ABB RobotStudio station: OP70 Robot Program.rspag

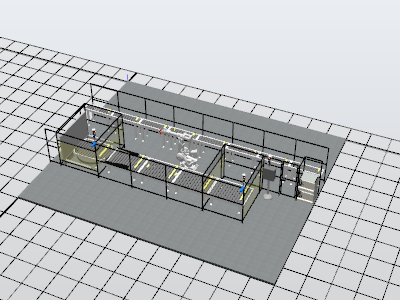
--- station ---
Station OP70 (saved by RobotStudio 24.3.10885.0)
Controller IRB4400_60_196_1, task T_ROB1: task frame (RAPID world) sits at (4963.29, 5843.46, 0) mm, rotated rx 0 ry 0 rz -90 deg in the station
Controller IRB4400_60_196_1
  mechanical unit ROB_1: IRB4400_60_196__03, 6 joints, base frame (0, 0, 0) mm
Layout (positions relative to the parent item):
  - Metal Floor 10 x 12 meter [part], size 10024.3 x 12025.3 x 126.6 mm
  - SOP710 [smart component] at (3750, 1320, 100) mm, rotated rx 0 ry 0 rz 90 deg
      properties: ForwardSpeed=0.05; ReverseSpeed=-0.05; ConveyorSpeed=0; SpeedForward=0.7; Constant=1E-09; SpeedBackward=-0.6
      signals: DI MotorFWD, DI MotorREV, DO ConveyorError, DI ResetError, DO MotorFeedback, DO BoxSensor
      connections:
        SOP710.MotorFWD -> ?.Enabled
        SOP710.MotorREV -> ?.Enabled
        ?.Output -> ?.Enabled
        SOP710.MotorFWD -> ?.Execute
        SOP710.MotorREV -> ?.Execute
        SOP710.MotorFWD -> ?.A
        SOP710.MotorREV -> ?.B
        ?.Result -> ConveyorSurfaceBehaviour.SurfaceVelocity
        ?.Output -> ConveyorSurfaceBehaviour.SurfaceVelocity
        ?.Output -> ?.InputA
        ?.Output -> ?.InputB
        SOP710.MotorFWD -> ?.InputA
        SOP710.MotorFWD -> ?.InputA
        SOP710.MotorREV -> ?.InputB
        SOP710.MotorFWD -> ?.InputA
        SOP710.MotorFWD -> ?.A
        ?.Result -> ConveyorSurfaceBehaviour.SurfaceVelocity
        SOP710.MotorFWD -> ?.Set
        SOP710.MotorREV -> ?.Set
        SetIdleSpeed.Result -> SetIdleSpeedToConveyor.Execute
        SOP710.MotorFWD -> SetIdleSpeed.A
        SOP710.MotorREV -> SetIdleSpeed.B
        SOP710.MotorFWD -> SetMotorSafetyBreaker.FWD
        SOP710.MotorREV -> SetMotorSafetyBreaker.REV
        ErrorCheckAndBlockingMotorsAndErrorResetLogic.Output -> SetIdleSpeedToConveyor.Execute
        SOP710.ResetError -> ErrorCheckAndBlockingMotorsAndErrorResetLogic.Reset
        SOP710.MotorFWD -> NoErrorAllowFWD.FWD
        ErrorCheckAndBlockingMotorsAndErrorResetLogic.Output -> NoErrorAllowFWD.Error
        NoErrorAllowFWD.Result -> SetForwardSpeedToConveyor.Execute
        SOP710.MotorREV -> NoErrorAllowREV.REV
        ErrorCheckAndBlockingMotorsAndErrorResetLogic.Output -> NoErrorAllowREV.Error
        NoErrorAllowREV.Result -> SetBackwardSpeedToConveyor.Execute
        SetMotorSafetyBreaker.Result -> ErrorCheckAndBlockingMotorsAndErrorResetLogic.Set
        GraphicsHideLogic.Result -> GraphicsHide.Execute
        SOP710.MotorFWD -> GraphicsHideLogic.FWD
        SOP710.MotorREV -> GraphicsHideLogic.REV
        SOP710.MotorFWD -> MotorFeedbackSignalLogic.A
        SOP710.MotorREV -> MotorFeedbackSignalLogic.A
        ErrorCheckAndBlockingMotorsAndErrorResetLogic.Output -> MotorFeedbackSignalLogic.B
        MotorFeedbackSignalLogic.Result -> SOP710.MotorFeedback
        MotorFeedbackSignalLogic.Result -> GraphicsShow.Execute
        ErrorCheckAndBlockingMotorsAndErrorResetLogic.InvOutput -> SOP710.ConveyorError
        SUB610_B1.SensorSignal -> SOP710.BoxSensor
        ?.Result => ?.Count
        ?.Value => ConveyorSurfaceBehaviour.SurfaceVelocity
        ?.Value => ConveyorSurfaceBehaviour.SurfaceVelocity
        ?.Value => ConveyorSurfaceBehaviour.SurfaceVelocity
        ?.Value => ConveyorSurfaceBehaviour.SurfaceVelocity
        ?.Value => ConveyorSurfaceBehaviour.SurfaceVelocity
        ?.Value => ConveyorSurfaceBehaviour.SurfaceVelocity
        SetIdleSpeedToConveyor.Value => ConveyorSurfaceBehaviour.SurfaceVelocity
        SetForwardSpeedToConveyor.Value => ConveyorSurfaceBehaviour.SurfaceVelocity
        SetBackwardSpeedToConveyor.Value => ConveyorSurfaceBehaviour.SurfaceVelocity
        ?.Result => SetForwardSpeedToConveyor.Max
        ?.A => SetBackwardSpeedToConveyor.Min
        ?.Result => SetBackwardSpeedToConveyor.Max
        ?.A => SetForwardSpeedToConveyor.Min
        GraphicsShow.Object => GraphicsHide.Object
        ?.Object => ?.Object
    - ConveyorSurfaceBehaviour [smart component, from Components\PhysicsControl.rslib] at (-701.82, -354.86, 903.18) mm
        properties: Object=ConveyorSurface; Behavior=1; SurfaceVelocity=0
    - SetIdleSpeedToConveyor [smart component, from Components\Random.rslib] at (-701.82, -354.86, 903.18) mm
        properties: Value=0; Min=0; Max=1E-13
    - SetBackwardSpeedToConveyor [smart component, from Components\Random.rslib] at (-701.82, -354.86, 903.18) mm
        properties: Value=-0.69999999999997; Min=-0.7; Max=-0.6999999999999
    - SetForwardSpeedToConveyor [smart component, from Components\Random.rslib] at (-701.82, -354.86, 903.18) mm
        properties: Value=0.500000000089343; Min=0.5; Max=0.5000000001
    - SetIdleSpeed [smart component, from Components\LogicExpression.rslib] at (-701.82, -354.86, 903.18) mm
        properties: Expression=not A and not B
    - SetMotorSafetyBreaker [smart component, from Components\LogicExpression.rslib] at (-701.82, -354.86, 903.18) mm
        properties: Expression=FWD and REV
    - ErrorCheckAndBlockingMotorsAndErrorResetLogic [smart component, from Components\LogicSRLatch.rslib] at (-701.82, -354.86, 903.18) mm
    - NoErrorAllowFWD [smart component, from Components\LogicExpression.rslib] at (-701.82, -354.86, 903.18) mm
        properties: Expression=FWD and not Error
    - NoErrorAllowREV [smart component, from Components\LogicExpression.rslib] at (-701.82, -354.86, 903.18) mm
        properties: Expression=REV and not Error
    - GraphicsShow [smart component, from Components\Show.rslib] at (-701.82, -354.86, 903.18) mm
        properties: Object=OnOffGfx
    - GraphicsHide [smart component, from Components\Hide.rslib] at (-701.82, -354.86, 903.18) mm
        properties: Object=OnOffGfx
    - GraphicsHideLogic [smart component, from Components\LogicExpression.rslib] at (-701.82, -354.86, 903.18) mm
        properties: Expression=not FWD and not REV
    - GraphicsObjects [graphiccomponentgroup] at (83.9, 149.37, 1003.18) mm, rotated rx 0 ry 0 rz -90 deg
      - OnOffGfx [graphiccomponentgroup] at (514.42, -850.96, -110.92) mm, rotated rx 0 ry 0 rz 90 deg
        - Part_5 [part] at (927.42, 264.29, 0) mm, rotated rx 0 ry 0 rz -90 deg, size 50 x 1493.5 x 100 mm
        - Part_6 [part] at (926.46, -134.61, 0) mm, rotated rx 0 ry 0 rz -90 deg, size 50 x 1492.5 x 100 mm
      - ConveyorSurface [part] at (-0.94, 65.23, -516.89) mm, rotated rx 0 ry 0 rz 180 deg, size 356.8 x 1451.8 x 107.9 mm
    - MotorFeedbackSignalLogic [smart component, from Components\LogicExpression.rslib] at (-701.82, -354.86, 903.18) mm
        properties: Expression=A AND NOT B
    - 1500x450x500 [graphiccomponentgroup] at (162.8, -49.34, 486.29) mm, rotated rx 0 ry 0 rz 180 deg
      - GeneratedPart [part] at (0, 0, 380) mm, size 1500 x 50 x 120 mm
      - GeneratedPart_2 [part] at (0, 400, 380) mm, size 1500 x 50 x 120 mm
      - GeneratedPart_3 [part] at (0, 50, 380) mm, size 50 x 350 x 120 mm
      - GeneratedPart_4 [part] at (1450, 50, 380) mm, size 50 x 350 x 120 mm
      - GeneratedPart_5 [part] at (150, 0, 72) mm
      - GeneratedPart_6 [part] at (150, 0, 72) mm
      - GeneratedPart_7 [part] at (150, 400, 72) mm
      - GeneratedPart_8 [part] at (125, 50, 460) mm, rotated rx -90 ry 0 rz 0 deg, size 80 x 79.7 x 350 mm
      - GeneratedPart_9 [part] at (162.5, -50, 0) mm
      - GeneratedPart_10 [part] at (162.5, -50, 0) mm
      - GeneratedPart_11 [part] at (162.5, 400, 0) mm
      - GeneratedPart_12 [part] at (125, 50, 460) mm, rotated rx -90 ry 0 rz 0 deg, size 80 x 79.7 x 350 mm
      - GeneratedPart_13 [part] at (250, 50, 460) mm, rotated rx -90 ry 0 rz 0 deg, size 80 x 79.7 x 350 mm
      - GeneratedPart_14 [part] at (375, 50, 460) mm, rotated rx -90 ry 0 rz 0 deg, size 80 x 79.7 x 350 mm
      - GeneratedPart_15 [part] at (500, 50, 460) mm, rotated rx -90 ry 0 rz 0 deg, size 80 x 79.7 x 350 mm
      - GeneratedPart_16 [part] at (625, 50, 460) mm, rotated rx -90 ry 0 rz 0 deg, size 80 x 79.7 x 350 mm
      - GeneratedPart_17 [part] at (750, 50, 460) mm, rotated rx -90 ry 0 rz 0 deg, size 80 x 79.7 x 350 mm
      - GeneratedPart_18 [part] at (875, 50, 460) mm, rotated rx -90 ry 0 rz 0 deg, size 80 x 79.7 x 350 mm
      - GeneratedPart_19 [part] at (1000, 50, 460) mm, rotated rx -90 ry 0 rz 0 deg, size 80 x 79.7 x 350 mm
      - GeneratedPart_20 [part] at (1125, 50, 460) mm, rotated rx -90 ry 0 rz 0 deg, size 80 x 79.7 x 350 mm
      - GeneratedPart_21 [part] at (1250, 50, 460) mm, rotated rx -90 ry 0 rz 0 deg, size 80 x 79.7 x 350 mm
      - GeneratedPart_22 [part] at (1375, 50, 460) mm, rotated rx -90 ry 0 rz 0 deg, size 80 x 79.7 x 350 mm
      - GeneratedPart_23 [part] at (200, 25, 12) mm
      - GeneratedPart_24 [part] at (200, 25, 12) mm
      - GeneratedPart_25 [part] at (200, 425, 12) mm
      - GeneratedPart_26 [part] at (1266.54, 400, 0) mm
      - GeneratedPart_27 [part] at (1254.04, 0, 72) mm
      - GeneratedPart_28 [part] at (1304.04, 25, 12) mm
      - GeneratedPart_29 [part] at (1266.54, -50, 0) mm
      - GeneratedPart_30 [part] at (1254.04, 400, 72) mm
      - GeneratedPart_31 [part] at (1304.04, 425, 12) mm
      - Part_3 [part] at (1105.7, 0.66, -486.29) mm, size 100 x 550 x 880 mm
      - Part_2 [part] at (0.3, 0.66, -486.29) mm, size 100 x 550 x 880 mm
    - SUB610_B1 [smart component] at (-13.16, -49.69, 870.13) mm, rotated rx 0 ry 0 rz 180 deg
        signals: DO SensorSignal
        connections:
          SensorRay.SensorOut -> ?.Active
          ?.Output -> SUB610_B1.SensorSignal
          SensorRay.SensorOut -> LogicGate.InputA
          GraphicSwitch_2.Output -> LogicGate_2.InputA
          LogicGate_2.Output -> LogicGate.InputB
          LogicGate.Output -> SUB610_B1.SensorSignal
      - SensorRay [smart component, from Components\LineSensor.rslib] at (24.04, 61.94, 174.13) mm
          properties: Start=[0 0 0]; End=[1.02087466601758E-07 0.23805885165687 4.04628539979468E-07]; Radius=0.01; SensedPart=(none); SensedPoint=[0 0 0]; Length=0.238058851657236; Tag=(none)
        - _sensorPart_ [part], size 20 x 238.1 x 20 mm
      - SensorMountWorking [part] at (0, 0, 0) mm, size 50 x 50 x 200 mm
      - GraphicSwitch_2 [smart component, from Components\GraphicSwitch.rslib] at (50, 0, 0) mm
          properties: PartHigh=SensorMountBroken; PartLow=SensorMountWorking
      - SensorMountBroken [part] at (0, 0, 0) mm, size 50 x 50 x 200 mm
      - LogicGate [smart component, from Components\LogicGate.rslib]
          properties: Operator=AND; Delay=0
      - LogicGate_2 [smart component, from Components\LogicGate.rslib]
          properties: Operator=NOT; Delay=0
  - SOP712 [smart component] at (3750, 4320, 100) mm, rotated rx 0 ry 0 rz 90 deg
      properties: ForwardSpeed=0.05; ReverseSpeed=-0.05; ConveyorSpeed=0; SpeedForward=0.7; Constant=1E-09; SpeedBackward=-0.6
      signals: DI MotorFWD, DI MotorREV, DO ConveyorError, DI ResetError, DO MotorFeedback, DO BoxSensor
      connections:
        SOP712.MotorFWD -> ?.Enabled
        SOP712.MotorREV -> ?.Enabled
        ?.Output -> ?.Enabled
        SOP712.MotorFWD -> ?.Execute
        SOP712.MotorREV -> ?.Execute
        SOP712.MotorFWD -> ?.A
        SOP712.MotorREV -> ?.B
        ?.Result -> ConveyorSurfaceBehaviour.SurfaceVelocity
        ?.Output -> ConveyorSurfaceBehaviour.SurfaceVelocity
        ?.Output -> ?.InputA
        ?.Output -> ?.InputB
        SOP712.MotorFWD -> ?.InputA
        SOP712.MotorFWD -> ?.InputA
        SOP712.MotorREV -> ?.InputB
        SOP712.MotorFWD -> ?.InputA
        SOP712.MotorFWD -> ?.A
        ?.Result -> ConveyorSurfaceBehaviour.SurfaceVelocity
        SOP712.MotorFWD -> ?.Set
        SOP712.MotorREV -> ?.Set
        SetIdleSpeed.Result -> SetIdleSpeedToConveyor.Execute
        SOP712.MotorFWD -> SetIdleSpeed.A
        SOP712.MotorREV -> SetIdleSpeed.B
        SOP712.MotorFWD -> SetMotorSafetyBreaker.FWD
        SOP712.MotorREV -> SetMotorSafetyBreaker.REV
        ErrorCheckAndBlockingMotorsAndErrorResetLogic.Output -> SetIdleSpeedToConveyor.Execute
        SOP712.ResetError -> ErrorCheckAndBlockingMotorsAndErrorResetLogic.Reset
        SOP712.MotorFWD -> NoErrorAllowFWD.FWD
        ErrorCheckAndBlockingMotorsAndErrorResetLogic.Output -> NoErrorAllowFWD.Error
        NoErrorAllowFWD.Result -> SetForwardSpeedToConveyor.Execute
        SOP712.MotorREV -> NoErrorAllowREV.REV
        ErrorCheckAndBlockingMotorsAndErrorResetLogic.Output -> NoErrorAllowREV.Error
        NoErrorAllowREV.Result -> SetBackwardSpeedToConveyor.Execute
        SetMotorSafetyBreaker.Result -> ErrorCheckAndBlockingMotorsAndErrorResetLogic.Set
        GraphicsHideLogic.Result -> GraphicsHide.Execute
        SOP712.MotorFWD -> GraphicsHideLogic.FWD
        SOP712.MotorREV -> GraphicsHideLogic.REV
        SOP712.MotorFWD -> MotorFeedbackSignalLogic.A
        SOP712.MotorREV -> MotorFeedbackSignalLogic.A
        ErrorCheckAndBlockingMotorsAndErrorResetLogic.Output -> MotorFeedbackSignalLogic.B
        MotorFeedbackSignalLogic.Result -> SOP712.MotorFeedback
        MotorFeedbackSignalLogic.Result -> GraphicsShow.Execute
        ErrorCheckAndBlockingMotorsAndErrorResetLogic.InvOutput -> SOP712.ConveyorError
        SUB610_B1.SensorSignal -> SOP712.BoxSensor
        ?.Result => ?.Count
        ?.Value => ConveyorSurfaceBehaviour.SurfaceVelocity
        ?.Value => ConveyorSurfaceBehaviour.SurfaceVelocity
        ?.Value => ConveyorSurfaceBehaviour.SurfaceVelocity
        ?.Value => ConveyorSurfaceBehaviour.SurfaceVelocity
        ?.Value => ConveyorSurfaceBehaviour.SurfaceVelocity
        ?.Value => ConveyorSurfaceBehaviour.SurfaceVelocity
        SetIdleSpeedToConveyor.Value => ConveyorSurfaceBehaviour.SurfaceVelocity
        SetForwardSpeedToConveyor.Value => ConveyorSurfaceBehaviour.SurfaceVelocity
        SetBackwardSpeedToConveyor.Value => ConveyorSurfaceBehaviour.SurfaceVelocity
        ?.Result => SetForwardSpeedToConveyor.Max
        ?.A => SetBackwardSpeedToConveyor.Min
        ?.Result => SetBackwardSpeedToConveyor.Max
        ?.A => SetForwardSpeedToConveyor.Min
        GraphicsShow.Object => GraphicsHide.Object
        ?.Object => ?.Object
    - ConveyorSurfaceBehaviour [smart component, from Components\PhysicsControl.rslib] at (-701.82, -354.86, 903.18) mm
        properties: Object=ConveyorSurface; Behavior=1; SurfaceVelocity=0
    - SetIdleSpeedToConveyor [smart component, from Components\Random.rslib] at (-701.82, -354.86, 903.18) mm
        properties: Value=0; Min=0; Max=1E-13
    - SetBackwardSpeedToConveyor [smart component, from Components\Random.rslib] at (-701.82, -354.86, 903.18) mm
        properties: Value=-0.69999999999993; Min=-0.7; Max=-0.6999999999999
    - SetForwardSpeedToConveyor [smart component, from Components\Random.rslib] at (-701.82, -354.86, 903.18) mm
        properties: Value=0.500000000032373; Min=0.5; Max=0.5000000001
    - SetIdleSpeed [smart component, from Components\LogicExpression.rslib] at (-701.82, -354.86, 903.18) mm
        properties: Expression=not A and not B
    - SetMotorSafetyBreaker [smart component, from Components\LogicExpression.rslib] at (-701.82, -354.86, 903.18) mm
        properties: Expression=FWD and REV
    - ErrorCheckAndBlockingMotorsAndErrorResetLogic [smart component, from Components\LogicSRLatch.rslib] at (-701.82, -354.86, 903.18) mm
    - NoErrorAllowFWD [smart component, from Components\LogicExpression.rslib] at (-701.82, -354.86, 903.18) mm
        properties: Expression=FWD and not Error
    - NoErrorAllowREV [smart component, from Components\LogicExpression.rslib] at (-701.82, -354.86, 903.18) mm
        properties: Expression=REV and not Error
    - GraphicsShow [smart component, from Components\Show.rslib] at (-701.82, -354.86, 903.18) mm
        properties: Object=OnOffGfx
    - GraphicsHide [smart component, from Components\Hide.rslib] at (-701.82, -354.86, 903.18) mm
        properties: Object=OnOffGfx
    - GraphicsHideLogic [smart component, from Components\LogicExpression.rslib] at (-701.82, -354.86, 903.18) mm
        properties: Expression=not FWD and not REV
    - GraphicsObjects [graphiccomponentgroup] at (83.9, 149.37, 1003.18) mm, rotated rx 0 ry 0 rz -90 deg
      - OnOffGfx [graphiccomponentgroup] at (514.42, -850.96, -110.92) mm, rotated rx 0 ry 0 rz 90 deg
        - Part_5 [part] at (927.42, 264.29, 0) mm, rotated rx 0 ry 0 rz -90 deg, size 50 x 1493.5 x 100 mm
        - Part_6 [part] at (926.46, -134.61, 0) mm, rotated rx 0 ry 0 rz -90 deg, size 50 x 1492.5 x 100 mm
      - ConveyorSurface [part] at (-0.94, 65.23, -516.89) mm, rotated rx 0 ry 0 rz 180 deg, size 356.8 x 1451.8 x 107.9 mm
    - MotorFeedbackSignalLogic [smart component, from Components\LogicExpression.rslib] at (-701.82, -354.86, 903.18) mm
        properties: Expression=A AND NOT B
    - 1500x450x500 [graphiccomponentgroup] at (162.8, -49.34, 486.29) mm, rotated rx 0 ry 0 rz 180 deg
      - GeneratedPart [part] at (0, 0, 380) mm, size 1500 x 50 x 120 mm
      - GeneratedPart_2 [part] at (0, 400, 380) mm, size 1500 x 50 x 120 mm
      - GeneratedPart_3 [part] at (0, 50, 380) mm, size 50 x 350 x 120 mm
      - GeneratedPart_4 [part] at (1450, 50, 380) mm, size 50 x 350 x 120 mm
      - GeneratedPart_5 [part] at (150, 0, 72) mm
      - GeneratedPart_6 [part] at (150, 0, 72) mm
      - GeneratedPart_7 [part] at (150, 400, 72) mm
      - GeneratedPart_8 [part] at (125, 50, 460) mm, rotated rx -90 ry 0 rz 0 deg, size 80 x 79.7 x 350 mm
      - GeneratedPart_9 [part] at (162.5, -50, 0) mm
      - GeneratedPart_10 [part] at (162.5, -50, 0) mm
      - GeneratedPart_11 [part] at (162.5, 400, 0) mm
      - GeneratedPart_12 [part] at (125, 50, 460) mm, rotated rx -90 ry 0 rz 0 deg, size 80 x 79.7 x 350 mm
      - GeneratedPart_13 [part] at (250, 50, 460) mm, rotated rx -90 ry 0 rz 0 deg, size 80 x 79.7 x 350 mm
      - GeneratedPart_14 [part] at (375, 50, 460) mm, rotated rx -90 ry 0 rz 0 deg, size 80 x 79.7 x 350 mm
      - GeneratedPart_15 [part] at (500, 50, 460) mm, rotated rx -90 ry 0 rz 0 deg, size 80 x 79.7 x 350 mm
      - GeneratedPart_16 [part] at (625, 50, 460) mm, rotated rx -90 ry 0 rz 0 deg, size 80 x 79.7 x 350 mm
      - GeneratedPart_17 [part] at (750, 50, 460) mm, rotated rx -90 ry 0 rz 0 deg, size 80 x 79.7 x 350 mm
      - GeneratedPart_18 [part] at (875, 50, 460) mm, rotated rx -90 ry 0 rz 0 deg, size 80 x 79.7 x 350 mm
      - GeneratedPart_19 [part] at (1000, 50, 460) mm, rotated rx -90 ry 0 rz 0 deg, size 80 x 79.7 x 350 mm
      - GeneratedPart_20 [part] at (1125, 50, 460) mm, rotated rx -90 ry 0 rz 0 deg, size 80 x 79.7 x 350 mm
      - GeneratedPart_21 [part] at (1250, 50, 460) mm, rotated rx -90 ry 0 rz 0 deg, size 80 x 79.7 x 350 mm
      - GeneratedPart_22 [part] at (1375, 50, 460) mm, rotated rx -90 ry 0 rz 0 deg, size 80 x 79.7 x 350 mm
      - GeneratedPart_23 [part] at (200, 25, 12) mm
      - GeneratedPart_24 [part] at (200, 25, 12) mm
      - GeneratedPart_25 [part] at (200, 425, 12) mm
      - GeneratedPart_26 [part] at (1266.54, 400, 0) mm
      - GeneratedPart_27 [part] at (1254.04, 0, 72) mm
      - GeneratedPart_28 [part] at (1304.04, 25, 12) mm
      - GeneratedPart_29 [part] at (1266.54, -50, 0) mm
      - GeneratedPart_30 [part] at (1254.04, 400, 72) mm
      - GeneratedPart_31 [part] at (1304.04, 425, 12) mm
      - Part_3 [part] at (1105.7, 0.66, -486.29) mm, size 100 x 550 x 880 mm
      - Part_2 [part] at (0.3, 0.66, -486.29) mm, size 100 x 550 x 880 mm
    - SUB610_B1 [smart component] at (-13.16, -49.69, 870.13) mm, rotated rx 0 ry 0 rz 180 deg
        signals: DO SensorSignal
        connections:
          SensorRay.SensorOut -> ?.Active
          ?.Output -> SUB610_B1.SensorSignal
          SensorRay.SensorOut -> LogicGate.InputA
          GraphicSwitch_2.Output -> LogicGate_2.InputA
          LogicGate_2.Output -> LogicGate.InputB
          LogicGate.Output -> SUB610_B1.SensorSignal
      - SensorRay [smart component, from Components\LineSensor.rslib] at (24.04, 61.94, 174.13) mm
          properties: Start=[0 0 0]; End=[1.02087466601758E-07 0.23805885165687 4.04628539979468E-07]; Radius=0.01; SensedPart=(none); SensedPoint=[0 0 0]; Length=0.238058851657236; Tag=(none)
        - _sensorPart_ [part], size 20 x 238.1 x 20 mm
      - SensorMountWorking [part] at (0, 0, 0) mm, size 50 x 50 x 200 mm
      - GraphicSwitch_2 [smart component, from Components\GraphicSwitch.rslib] at (50, 0, 0) mm
          properties: PartHigh=SensorMountBroken; PartLow=SensorMountWorking
      - SensorMountBroken [part] at (0, 0, 0) mm, size 50 x 50 x 200 mm
      - LogicGate [smart component, from Components\LogicGate.rslib]
          properties: Operator=AND; Delay=0
      - LogicGate_2 [smart component, from Components\LogicGate.rslib]
          properties: Operator=NOT; Delay=0
  - SOP711 [smart component] at (3750, 2820, 100) mm, rotated rx 0 ry 0 rz 90 deg
      properties: ForwardSpeed=0.05; ReverseSpeed=-0.05; ConveyorSpeed=0; SpeedForward=0.7; Constant=1E-09; SpeedBackward=-0.6
      signals: DI MotorFWD, DI MotorREV, DO ConveyorError, DI ResetError, DO MotorFeedback, DO BoxSensor
      connections:
        SOP711.MotorFWD -> ?.Enabled
        SOP711.MotorREV -> ?.Enabled
        ?.Output -> ?.Enabled
        SOP711.MotorFWD -> ?.Execute
        SOP711.MotorREV -> ?.Execute
        SOP711.MotorFWD -> ?.A
        SOP711.MotorREV -> ?.B
        ?.Result -> ConveyorSurfaceBehaviour.SurfaceVelocity
        ?.Output -> ConveyorSurfaceBehaviour.SurfaceVelocity
        ?.Output -> ?.InputA
        ?.Output -> ?.InputB
        SOP711.MotorFWD -> ?.InputA
        SOP711.MotorFWD -> ?.InputA
        SOP711.MotorREV -> ?.InputB
        SOP711.MotorFWD -> ?.InputA
        SOP711.MotorFWD -> ?.A
        ?.Result -> ConveyorSurfaceBehaviour.SurfaceVelocity
        SOP711.MotorFWD -> ?.Set
        SOP711.MotorREV -> ?.Set
        SetIdleSpeed.Result -> SetIdleSpeedToConveyor.Execute
        SOP711.MotorFWD -> SetIdleSpeed.A
        SOP711.MotorREV -> SetIdleSpeed.B
        SOP711.MotorFWD -> SetMotorSafetyBreaker.FWD
        SOP711.MotorREV -> SetMotorSafetyBreaker.REV
        ErrorCheckAndBlockingMotorsAndErrorResetLogic.Output -> SetIdleSpeedToConveyor.Execute
        SOP711.ResetError -> ErrorCheckAndBlockingMotorsAndErrorResetLogic.Reset
        SOP711.MotorFWD -> NoErrorAllowFWD.FWD
        ErrorCheckAndBlockingMotorsAndErrorResetLogic.Output -> NoErrorAllowFWD.Error
        NoErrorAllowFWD.Result -> SetForwardSpeedToConveyor.Execute
        SOP711.MotorREV -> NoErrorAllowREV.REV
        ErrorCheckAndBlockingMotorsAndErrorResetLogic.Output -> NoErrorAllowREV.Error
        NoErrorAllowREV.Result -> SetBackwardSpeedToConveyor.Execute
        SetMotorSafetyBreaker.Result -> ErrorCheckAndBlockingMotorsAndErrorResetLogic.Set
        GraphicsHideLogic.Result -> GraphicsHide.Execute
        SOP711.MotorFWD -> GraphicsHideLogic.FWD
        SOP711.MotorREV -> GraphicsHideLogic.REV
        SOP711.MotorFWD -> MotorFeedbackSignalLogic.A
        SOP711.MotorREV -> MotorFeedbackSignalLogic.A
        ErrorCheckAndBlockingMotorsAndErrorResetLogic.Output -> MotorFeedbackSignalLogic.B
        MotorFeedbackSignalLogic.Result -> SOP711.MotorFeedback
        MotorFeedbackSignalLogic.Result -> GraphicsShow.Execute
        ErrorCheckAndBlockingMotorsAndErrorResetLogic.InvOutput -> SOP711.ConveyorError
        SUB610_B1.SensorSignal -> SOP711.BoxSensor
        ?.Result => ?.Count
        ?.Value => ConveyorSurfaceBehaviour.SurfaceVelocity
        ?.Value => ConveyorSurfaceBehaviour.SurfaceVelocity
        ?.Value => ConveyorSurfaceBehaviour.SurfaceVelocity
        ?.Value => ConveyorSurfaceBehaviour.SurfaceVelocity
        ?.Value => ConveyorSurfaceBehaviour.SurfaceVelocity
        ?.Value => ConveyorSurfaceBehaviour.SurfaceVelocity
        SetIdleSpeedToConveyor.Value => ConveyorSurfaceBehaviour.SurfaceVelocity
        SetForwardSpeedToConveyor.Value => ConveyorSurfaceBehaviour.SurfaceVelocity
        SetBackwardSpeedToConveyor.Value => ConveyorSurfaceBehaviour.SurfaceVelocity
        ?.Result => SetForwardSpeedToConveyor.Max
        ?.A => SetBackwardSpeedToConveyor.Min
        ?.Result => SetBackwardSpeedToConveyor.Max
        ?.A => SetForwardSpeedToConveyor.Min
        GraphicsShow.Object => GraphicsHide.Object
        ?.Object => ?.Object
    - ConveyorSurfaceBehaviour [smart component, from Components\PhysicsControl.rslib] at (-701.82, -354.86, 903.18) mm
        properties: Object=ConveyorSurface; Behavior=1; SurfaceVelocity=7.88691123383442E-14
    - SetIdleSpeedToConveyor [smart component, from Components\Random.rslib] at (-701.82, -354.86, 903.18) mm
        properties: Value=7.88691123383442E-14; Min=0; Max=1E-13
    - SetBackwardSpeedToConveyor [smart component, from Components\Random.rslib] at (-701.82, -354.86, 903.18) mm
        properties: Value=-0.69999999999997; Min=-0.7; Max=-0.6999999999999
    - SetForwardSpeedToConveyor [smart component, from Components\Random.rslib] at (-701.82, -354.86, 903.18) mm
        properties: Value=0.500000000007179; Min=0.5; Max=0.5000000001
    - SetIdleSpeed [smart component, from Components\LogicExpression.rslib] at (-701.82, -354.86, 903.18) mm
        properties: Expression=not A and not B
    - SetMotorSafetyBreaker [smart component, from Components\LogicExpression.rslib] at (-701.82, -354.86, 903.18) mm
        properties: Expression=FWD and REV
    - ErrorCheckAndBlockingMotorsAndErrorResetLogic [smart component, from Components\LogicSRLatch.rslib] at (-701.82, -354.86, 903.18) mm
    - NoErrorAllowFWD [smart component, from Components\LogicExpression.rslib] at (-701.82, -354.86, 903.18) mm
        properties: Expression=FWD and not Error
    - NoErrorAllowREV [smart component, from Components\LogicExpression.rslib] at (-701.82, -354.86, 903.18) mm
        properties: Expression=REV and not Error
    - GraphicsShow [smart component, from Components\Show.rslib] at (-701.82, -354.86, 903.18) mm
        properties: Object=OnOffGfx
    - GraphicsHide [smart component, from Components\Hide.rslib] at (-701.82, -354.86, 903.18) mm
        properties: Object=OnOffGfx
    - GraphicsHideLogic [smart component, from Components\LogicExpression.rslib] at (-701.82, -354.86, 903.18) mm
        properties: Expression=not FWD and not REV
    - GraphicsObjects [graphiccomponentgroup] at (83.9, 149.37, 1003.18) mm, rotated rx 0 ry 0 rz -90 deg
      - OnOffGfx [graphiccomponentgroup] at (514.42, -850.96, -110.92) mm, rotated rx 0 ry 0 rz 90 deg
        - Part_5 [part] at (927.42, 264.29, 0) mm, rotated rx 0 ry 0 rz -90 deg, size 50 x 1493.5 x 100 mm
        - Part_6 [part] at (926.46, -134.61, 0) mm, rotated rx 0 ry 0 rz -90 deg, size 50 x 1492.5 x 100 mm
      - ConveyorSurface [part] at (-0.94, 65.23, -516.89) mm, rotated rx 0 ry 0 rz 180 deg, size 356.8 x 1451.8 x 107.9 mm
    - MotorFeedbackSignalLogic [smart component, from Components\LogicExpression.rslib] at (-701.82, -354.86, 903.18) mm
        properties: Expression=A AND NOT B
    - 1500x450x500 [graphiccomponentgroup] at (162.8, -49.34, 486.29) mm, rotated rx 0 ry 0 rz 180 deg
      - GeneratedPart [part] at (0, 0, 380) mm, size 1500 x 50 x 120 mm
      - GeneratedPart_2 [part] at (0, 400, 380) mm, size 1500 x 50 x 120 mm
      - GeneratedPart_3 [part] at (0, 50, 380) mm, size 50 x 350 x 120 mm
      - GeneratedPart_4 [part] at (1450, 50, 380) mm, size 50 x 350 x 120 mm
      - GeneratedPart_5 [part] at (150, 0, 72) mm
      - GeneratedPart_6 [part] at (150, 0, 72) mm
      - GeneratedPart_7 [part] at (150, 400, 72) mm
      - GeneratedPart_8 [part] at (125, 50, 460) mm, rotated rx -90 ry 0 rz 0 deg, size 80 x 79.7 x 350 mm
      - GeneratedPart_9 [part] at (162.5, -50, 0) mm
      - GeneratedPart_10 [part] at (162.5, -50, 0) mm
      - GeneratedPart_11 [part] at (162.5, 400, 0) mm
      - GeneratedPart_12 [part] at (125, 50, 460) mm, rotated rx -90 ry 0 rz 0 deg, size 80 x 79.7 x 350 mm
      - GeneratedPart_13 [part] at (250, 50, 460) mm, rotated rx -90 ry 0 rz 0 deg, size 80 x 79.7 x 350 mm
      - GeneratedPart_14 [part] at (375, 50, 460) mm, rotated rx -90 ry 0 rz 0 deg, size 80 x 79.7 x 350 mm
      - GeneratedPart_15 [part] at (500, 50, 460) mm, rotated rx -90 ry 0 rz 0 deg, size 80 x 79.7 x 350 mm
      - GeneratedPart_16 [part] at (625, 50, 460) mm, rotated rx -90 ry 0 rz 0 deg, size 80 x 79.7 x 350 mm
      - GeneratedPart_17 [part] at (750, 50, 460) mm, rotated rx -90 ry 0 rz 0 deg, size 80 x 79.7 x 350 mm
      - GeneratedPart_18 [part] at (875, 50, 460) mm, rotated rx -90 ry 0 rz 0 deg, size 80 x 79.7 x 350 mm
      - GeneratedPart_19 [part] at (1000, 50, 460) mm, rotated rx -90 ry 0 rz 0 deg, size 80 x 79.7 x 350 mm
      - GeneratedPart_20 [part] at (1125, 50, 460) mm, rotated rx -90 ry 0 rz 0 deg, size 80 x 79.7 x 350 mm
      - GeneratedPart_21 [part] at (1250, 50, 460) mm, rotated rx -90 ry 0 rz 0 deg, size 80 x 79.7 x 350 mm
      - GeneratedPart_22 [part] at (1375, 50, 460) mm, rotated rx -90 ry 0 rz 0 deg, size 80 x 79.7 x 350 mm
      - GeneratedPart_23 [part] at (200, 25, 12) mm
      - GeneratedPart_24 [part] at (200, 25, 12) mm
      - GeneratedPart_25 [part] at (200, 425, 12) mm
      - GeneratedPart_26 [part] at (1266.54, 400, 0) mm
      - GeneratedPart_27 [part] at (1254.04, 0, 72) mm
      - GeneratedPart_28 [part] at (1304.04, 25, 12) mm
      - GeneratedPart_29 [part] at (1266.54, -50, 0) mm
      - GeneratedPart_30 [part] at (1254.04, 400, 72) mm
      - GeneratedPart_31 [part] at (1304.04, 425, 12) mm
      - Part_3 [part] at (1105.7, 0.66, -486.29) mm, size 100 x 550 x 880 mm
      - Part_2 [part] at (0.3, 0.66, -486.29) mm, size 100 x 550 x 880 mm
    - SUB610_B1 [smart component] at (-13.16, -49.69, 870.13) mm, rotated rx 0 ry 0 rz 180 deg
        signals: DO SensorSignal
        connections:
          SensorRay.SensorOut -> ?.Active
          ?.Output -> SUB610_B1.SensorSignal
          SensorRay.SensorOut -> LogicGate.InputA
          GraphicSwitch_2.Output -> LogicGate_2.InputA
          LogicGate_2.Output -> LogicGate.InputB
          LogicGate.Output -> SUB610_B1.SensorSignal
      - SensorRay [smart component, from Components\LineSensor.rslib] at (24.04, 61.94, 174.13) mm
          properties: Start=[0 0 0]; End=[1.02087466601758E-07 0.23805885165687 4.04628539979468E-07]; Radius=0.01; SensedPart=(none); SensedPoint=[0 0 0]; Length=0.238058851657236; Tag=(none)
        - _sensorPart_ [part], size 20 x 238.1 x 20 mm
      - SensorMountWorking [part] at (0, 0, 0) mm, size 50 x 50 x 200 mm
      - GraphicSwitch_2 [smart component, from Components\GraphicSwitch.rslib] at (50, 0, 0) mm
          properties: PartHigh=SensorMountBroken; PartLow=SensorMountWorking
      - SensorMountBroken [part] at (0, 0, 0) mm, size 50 x 50 x 200 mm
      - LogicGate [smart component, from Components\LogicGate.rslib]
          properties: Operator=AND; Delay=0
      - LogicGate_2 [smart component, from Components\LogicGate.rslib]
          properties: Operator=NOT; Delay=0
  - SOP714 [smart component] at (3750, 7320, 100) mm, rotated rx 0 ry 0 rz 90 deg
      properties: ForwardSpeed=0.05; ReverseSpeed=-0.05; ConveyorSpeed=0; SpeedForward=0.7; Constant=1E-09; SpeedBackward=-0.6
      signals: DI MotorFWD, DI MotorREV, DO ConveyorError, DI ResetError, DO MotorFeedback, DO BoxSensor
      connections:
        SOP714.MotorFWD -> ?.Enabled
        SOP714.MotorREV -> ?.Enabled
        ?.Output -> ?.Enabled
        SOP714.MotorFWD -> ?.Execute
        SOP714.MotorREV -> ?.Execute
        SOP714.MotorFWD -> ?.A
        SOP714.MotorREV -> ?.B
        ?.Result -> ConveyorSurfaceBehaviour.SurfaceVelocity
        ?.Output -> ConveyorSurfaceBehaviour.SurfaceVelocity
        ?.Output -> ?.InputA
        ?.Output -> ?.InputB
        SOP714.MotorFWD -> ?.InputA
        SOP714.MotorFWD -> ?.InputA
        SOP714.MotorREV -> ?.InputB
        SOP714.MotorFWD -> ?.InputA
        SOP714.MotorFWD -> ?.A
        ?.Result -> ConveyorSurfaceBehaviour.SurfaceVelocity
        SOP714.MotorFWD -> ?.Set
        SOP714.MotorREV -> ?.Set
        SetIdleSpeed.Result -> SetIdleSpeedToConveyor.Execute
        SOP714.MotorFWD -> SetIdleSpeed.A
        SOP714.MotorREV -> SetIdleSpeed.B
        SOP714.MotorFWD -> SetMotorSafetyBreaker.FWD
        SOP714.MotorREV -> SetMotorSafetyBreaker.REV
        ErrorCheckAndBlockingMotorsAndErrorResetLogic.Output -> SetIdleSpeedToConveyor.Execute
        SOP714.ResetError -> ErrorCheckAndBlockingMotorsAndErrorResetLogic.Reset
        SOP714.MotorFWD -> NoErrorAllowFWD.FWD
        ErrorCheckAndBlockingMotorsAndErrorResetLogic.Output -> NoErrorAllowFWD.Error
        NoErrorAllowFWD.Result -> SetForwardSpeedToConveyor.Execute
        SOP714.MotorREV -> NoErrorAllowREV.REV
        ErrorCheckAndBlockingMotorsAndErrorResetLogic.Output -> NoErrorAllowREV.Error
        NoErrorAllowREV.Result -> SetBackwardSpeedToConveyor.Execute
        SetMotorSafetyBreaker.Result -> ErrorCheckAndBlockingMotorsAndErrorResetLogic.Set
        GraphicsHideLogic.Result -> GraphicsHide.Execute
        SOP714.MotorFWD -> GraphicsHideLogic.FWD
        SOP714.MotorREV -> GraphicsHideLogic.REV
        SOP714.MotorFWD -> MotorFeedbackSignalLogic.A
        SOP714.MotorREV -> MotorFeedbackSignalLogic.A
        ErrorCheckAndBlockingMotorsAndErrorResetLogic.Output -> MotorFeedbackSignalLogic.B
        MotorFeedbackSignalLogic.Result -> SOP714.MotorFeedback
        MotorFeedbackSignalLogic.Result -> GraphicsShow.Execute
        ErrorCheckAndBlockingMotorsAndErrorResetLogic.InvOutput -> SOP714.ConveyorError
        SUB610_B1.SensorSignal -> SOP714.BoxSensor
        ?.Result => ?.Count
        ?.Value => ConveyorSurfaceBehaviour.SurfaceVelocity
        ?.Value => ConveyorSurfaceBehaviour.SurfaceVelocity
        ?.Value => ConveyorSurfaceBehaviour.SurfaceVelocity
        ?.Value => ConveyorSurfaceBehaviour.SurfaceVelocity
        ?.Value => ConveyorSurfaceBehaviour.SurfaceVelocity
        ?.Value => ConveyorSurfaceBehaviour.SurfaceVelocity
        SetIdleSpeedToConveyor.Value => ConveyorSurfaceBehaviour.SurfaceVelocity
        SetForwardSpeedToConveyor.Value => ConveyorSurfaceBehaviour.SurfaceVelocity
        SetBackwardSpeedToConveyor.Value => ConveyorSurfaceBehaviour.SurfaceVelocity
        ?.Result => SetForwardSpeedToConveyor.Max
        ?.A => SetBackwardSpeedToConveyor.Min
        ?.Result => SetBackwardSpeedToConveyor.Max
        ?.A => SetForwardSpeedToConveyor.Min
        GraphicsShow.Object => GraphicsHide.Object
        ?.Object => ?.Object
    - ConveyorSurfaceBehaviour [smart component, from Components\PhysicsControl.rslib] at (-701.82, -354.86, 903.18) mm
        properties: Object=ConveyorSurface; Behavior=1; SurfaceVelocity=5.97368500939276E-14
    - SetIdleSpeedToConveyor [smart component, from Components\Random.rslib] at (-701.82, -354.86, 903.18) mm
        properties: Value=5.97368500939276E-14; Min=0; Max=1E-13
    - SetBackwardSpeedToConveyor [smart component, from Components\Random.rslib] at (-701.82, -354.86, 903.18) mm
        properties: Value=-0.69999999999997; Min=-0.7; Max=-0.6999999999999
    - SetForwardSpeedToConveyor [smart component, from Components\Random.rslib] at (-701.82, -354.86, 903.18) mm
        properties: Value=0.500000000073589; Min=0.5; Max=0.5000000001
    - SetIdleSpeed [smart component, from Components\LogicExpression.rslib] at (-701.82, -354.86, 903.18) mm
        properties: Expression=not A and not B
    - SetMotorSafetyBreaker [smart component, from Components\LogicExpression.rslib] at (-701.82, -354.86, 903.18) mm
        properties: Expression=FWD and REV
    - ErrorCheckAndBlockingMotorsAndErrorResetLogic [smart component, from Components\LogicSRLatch.rslib] at (-701.82, -354.86, 903.18) mm
    - NoErrorAllowFWD [smart component, from Components\LogicExpression.rslib] at (-701.82, -354.86, 903.18) mm
        properties: Expression=FWD and not Error
    - NoErrorAllowREV [smart component, from Components\LogicExpression.rslib] at (-701.82, -354.86, 903.18) mm
        properties: Expression=REV and not Error
    - GraphicsShow [smart component, from Components\Show.rslib] at (-701.82, -354.86, 903.18) mm
        properties: Object=OnOffGfx
    - GraphicsHide [smart component, from Components\Hide.rslib] at (-701.82, -354.86, 903.18) mm
        properties: Object=OnOffGfx
    - GraphicsHideLogic [smart component, from Components\LogicExpression.rslib] at (-701.82, -354.86, 903.18) mm
        properties: Expression=not FWD and not REV
    - GraphicsObjects [graphiccomponentgroup] at (83.9, 149.37, 1003.18) mm, rotated rx 0 ry 0 rz -90 deg
      - OnOffGfx [graphiccomponentgroup] at (514.42, -850.96, -110.92) mm, rotated rx 0 ry 0 rz 90 deg
        - Part_5 [part] at (927.42, 264.29, 0) mm, rotated rx 0 ry 0 rz -90 deg, size 50 x 1493.5 x 100 mm
        - Part_6 [part] at (926.46, -134.61, 0) mm, rotated rx 0 ry 0 rz -90 deg, size 50 x 1492.5 x 100 mm
      - ConveyorSurface [part] at (-0.94, 65.23, -516.89) mm, rotated rx 0 ry 0 rz 180 deg, size 356.8 x 1451.8 x 107.9 mm
    - MotorFeedbackSignalLogic [smart component, from Components\LogicExpression.rslib] at (-701.82, -354.86, 903.18) mm
        properties: Expression=A AND NOT B
    - 1500x450x500 [graphiccomponentgroup] at (162.8, -49.34, 486.29) mm, rotated rx 0 ry 0 rz 180 deg
      - GeneratedPart [part] at (0, 0, 380) mm, size 1500 x 50 x 120 mm
      - GeneratedPart_2 [part] at (0, 400, 380) mm, size 1500 x 50 x 120 mm
      - GeneratedPart_3 [part] at (0, 50, 380) mm, size 50 x 350 x 120 mm
      - GeneratedPart_4 [part] at (1450, 50, 380) mm, size 50 x 350 x 120 mm
      - GeneratedPart_5 [part] at (150, 0, 72) mm
      - GeneratedPart_6 [part] at (150, 0, 72) mm
      - GeneratedPart_7 [part] at (150, 400, 72) mm
      - GeneratedPart_8 [part] at (125, 50, 460) mm, rotated rx -90 ry 0 rz 0 deg, size 80 x 79.7 x 350 mm
      - GeneratedPart_9 [part] at (162.5, -50, 0) mm
      - GeneratedPart_10 [part] at (162.5, -50, 0) mm
      - GeneratedPart_11 [part] at (162.5, 400, 0) mm
      - GeneratedPart_12 [part] at (125, 50, 460) mm, rotated rx -90 ry 0 rz 0 deg, size 80 x 79.7 x 350 mm
      - GeneratedPart_13 [part] at (250, 50, 460) mm, rotated rx -90 ry 0 rz 0 deg, size 80 x 79.7 x 350 mm
      - GeneratedPart_14 [part] at (375, 50, 460) mm, rotated rx -90 ry 0 rz 0 deg, size 80 x 79.7 x 350 mm
      - GeneratedPart_15 [part] at (500, 50, 460) mm, rotated rx -90 ry 0 rz 0 deg, size 80 x 79.7 x 350 mm
      - GeneratedPart_16 [part] at (625, 50, 460) mm, rotated rx -90 ry 0 rz 0 deg, size 80 x 79.7 x 350 mm
      - GeneratedPart_17 [part] at (750, 50, 460) mm, rotated rx -90 ry 0 rz 0 deg, size 80 x 79.7 x 350 mm
      - GeneratedPart_18 [part] at (875, 50, 460) mm, rotated rx -90 ry 0 rz 0 deg, size 80 x 79.7 x 350 mm
      - GeneratedPart_19 [part] at (1000, 50, 460) mm, rotated rx -90 ry 0 rz 0 deg, size 80 x 79.7 x 350 mm
      - GeneratedPart_20 [part] at (1125, 50, 460) mm, rotated rx -90 ry 0 rz 0 deg, size 80 x 79.7 x 350 mm
      - GeneratedPart_21 [part] at (1250, 50, 460) mm, rotated rx -90 ry 0 rz 0 deg, size 80 x 79.7 x 350 mm
      - GeneratedPart_22 [part] at (1375, 50, 460) mm, rotated rx -90 ry 0 rz 0 deg, size 80 x 79.7 x 350 mm
      - GeneratedPart_23 [part] at (200, 25, 12) mm
      - GeneratedPart_24 [part] at (200, 25, 12) mm
      - GeneratedPart_25 [part] at (200, 425, 12) mm
      - GeneratedPart_26 [part] at (1266.54, 400, 0) mm
      - GeneratedPart_27 [part] at (1254.04, 0, 72) mm
      - GeneratedPart_28 [part] at (1304.04, 25, 12) mm
      - GeneratedPart_29 [part] at (1266.54, -50, 0) mm
      - GeneratedPart_30 [part] at (1254.04, 400, 72) mm
      - GeneratedPart_31 [part] at (1304.04, 425, 12) mm
      - Part_3 [part] at (1105.7, 0.66, -486.29) mm, size 100 x 550 x 880 mm
      - Part_2 [part] at (0.3, 0.66, -486.29) mm, size 100 x 550 x 880 mm
    - SUB610_B1 [smart component] at (-13.16, -49.69, 870.13) mm, rotated rx 0 ry 0 rz 180 deg
        signals: DO SensorSignal
        connections:
          SensorRay.SensorOut -> ?.Active
          ?.Output -> SUB610_B1.SensorSignal
          SensorRay.SensorOut -> LogicGate.InputA
          GraphicSwitch_2.Output -> LogicGate_2.InputA
          LogicGate_2.Output -> LogicGate.InputB
          LogicGate.Output -> SUB610_B1.SensorSignal
      - SensorRay [smart component, from Components\LineSensor.rslib] at (24.04, 61.94, 174.13) mm
          properties: Start=[0 0 0]; End=[1.02087466601758E-07 0.23805885165687 4.04628539979468E-07]; Radius=0.01; SensedPart=(none); SensedPoint=[0 0 0]; Length=0.238058851657236; Tag=(none)
        - _sensorPart_ [part], size 20 x 238.1 x 20 mm
      - SensorMountWorking [part] at (0, 0, 0) mm, size 50 x 50 x 200 mm
      - GraphicSwitch_2 [smart component, from Components\GraphicSwitch.rslib] at (50, 0, 0) mm
          properties: PartHigh=SensorMountBroken; PartLow=SensorMountWorking
      - SensorMountBroken [part] at (0, 0, 0) mm, size 50 x 50 x 200 mm
      - LogicGate [smart component, from Components\LogicGate.rslib]
          properties: Operator=AND; Delay=0
      - LogicGate_2 [smart component, from Components\LogicGate.rslib]
          properties: Operator=NOT; Delay=0
  - SOP715 [smart component] at (3750, 8820, 100) mm, rotated rx 0 ry 0 rz 90 deg
      properties: ForwardSpeed=0.05; ReverseSpeed=-0.05; ConveyorSpeed=0; SpeedForward=0.7; Constant=1E-09; SpeedBackward=-0.6
      signals: DI MotorFWD, DI MotorREV, DO ConveyorError, DI ResetError, DO MotorFeedback, DO BoxSensor
      connections:
        SOP715.MotorFWD -> ?.Enabled
        SOP715.MotorREV -> ?.Enabled
        ?.Output -> ?.Enabled
        SOP715.MotorFWD -> ?.Execute
        SOP715.MotorREV -> ?.Execute
        SOP715.MotorFWD -> ?.A
        SOP715.MotorREV -> ?.B
        ?.Result -> ConveyorSurfaceBehaviour.SurfaceVelocity
        ?.Output -> ConveyorSurfaceBehaviour.SurfaceVelocity
        ?.Output -> ?.InputA
        ?.Output -> ?.InputB
        SOP715.MotorFWD -> ?.InputA
        SOP715.MotorFWD -> ?.InputA
        SOP715.MotorREV -> ?.InputB
        SOP715.MotorFWD -> ?.InputA
        SOP715.MotorFWD -> ?.A
        ?.Result -> ConveyorSurfaceBehaviour.SurfaceVelocity
        SOP715.MotorFWD -> ?.Set
        SOP715.MotorREV -> ?.Set
        SetIdleSpeed.Result -> SetIdleSpeedToConveyor.Execute
        SOP715.MotorFWD -> SetIdleSpeed.A
        SOP715.MotorREV -> SetIdleSpeed.B
        SOP715.MotorFWD -> SetMotorSafetyBreaker.FWD
        SOP715.MotorREV -> SetMotorSafetyBreaker.REV
        ErrorCheckAndBlockingMotorsAndErrorResetLogic.Output -> SetIdleSpeedToConveyor.Execute
        SOP715.ResetError -> ErrorCheckAndBlockingMotorsAndErrorResetLogic.Reset
        SOP715.MotorFWD -> NoErrorAllowFWD.FWD
        ErrorCheckAndBlockingMotorsAndErrorResetLogic.Output -> NoErrorAllowFWD.Error
        NoErrorAllowFWD.Result -> SetForwardSpeedToConveyor.Execute
        SOP715.MotorREV -> NoErrorAllowREV.REV
        ErrorCheckAndBlockingMotorsAndErrorResetLogic.Output -> NoErrorAllowREV.Error
        NoErrorAllowREV.Result -> SetBackwardSpeedToConveyor.Execute
        SetMotorSafetyBreaker.Result -> ErrorCheckAndBlockingMotorsAndErrorResetLogic.Set
        GraphicsHideLogic.Result -> GraphicsHide.Execute
        SOP715.MotorFWD -> GraphicsHideLogic.FWD
        SOP715.MotorREV -> GraphicsHideLogic.REV
        SOP715.MotorFWD -> MotorFeedbackSignalLogic.A
        SOP715.MotorREV -> MotorFeedbackSignalLogic.A
        ErrorCheckAndBlockingMotorsAndErrorResetLogic.Output -> MotorFeedbackSignalLogic.B
        MotorFeedbackSignalLogic.Result -> SOP715.MotorFeedback
        MotorFeedbackSignalLogic.Result -> GraphicsShow.Execute
        ErrorCheckAndBlockingMotorsAndErrorResetLogic.InvOutput -> SOP715.ConveyorError
        SUB610_B1.SensorSignal -> SOP715.BoxSensor
        ?.Result => ?.Count
        ?.Value => ConveyorSurfaceBehaviour.SurfaceVelocity
        ?.Value => ConveyorSurfaceBehaviour.SurfaceVelocity
        ?.Value => ConveyorSurfaceBehaviour.SurfaceVelocity
        ?.Value => ConveyorSurfaceBehaviour.SurfaceVelocity
        ?.Value => ConveyorSurfaceBehaviour.SurfaceVelocity
        ?.Value => ConveyorSurfaceBehaviour.SurfaceVelocity
        SetIdleSpeedToConveyor.Value => ConveyorSurfaceBehaviour.SurfaceVelocity
        SetForwardSpeedToConveyor.Value => ConveyorSurfaceBehaviour.SurfaceVelocity
        SetBackwardSpeedToConveyor.Value => ConveyorSurfaceBehaviour.SurfaceVelocity
        ?.Result => SetForwardSpeedToConveyor.Max
        ?.A => SetBackwardSpeedToConveyor.Min
        ?.Result => SetBackwardSpeedToConveyor.Max
        ?.A => SetForwardSpeedToConveyor.Min
        GraphicsShow.Object => GraphicsHide.Object
        ?.Object => ?.Object
    - ConveyorSurfaceBehaviour [smart component, from Components\PhysicsControl.rslib] at (-701.82, -354.86, 903.18) mm
        properties: Object=ConveyorSurface; Behavior=1; SurfaceVelocity=5.48375129489403E-14
    - SetIdleSpeedToConveyor [smart component, from Components\Random.rslib] at (-701.82, -354.86, 903.18) mm
        properties: Value=5.48375129489403E-14; Min=0; Max=1E-13
    - SetBackwardSpeedToConveyor [smart component, from Components\Random.rslib] at (-701.82, -354.86, 903.18) mm
        properties: Value=-0.69999999999997; Min=-0.7; Max=-0.6999999999999
    - SetForwardSpeedToConveyor [smart component, from Components\Random.rslib] at (-701.82, -354.86, 903.18) mm
        properties: Value=0.500000000041715; Min=0.5; Max=0.5000000001
    - SetIdleSpeed [smart component, from Components\LogicExpression.rslib] at (-701.82, -354.86, 903.18) mm
        properties: Expression=not A and not B
    - SetMotorSafetyBreaker [smart component, from Components\LogicExpression.rslib] at (-701.82, -354.86, 903.18) mm
        properties: Expression=FWD and REV
    - ErrorCheckAndBlockingMotorsAndErrorResetLogic [smart component, from Components\LogicSRLatch.rslib] at (-701.82, -354.86, 903.18) mm
    - NoErrorAllowFWD [smart component, from Components\LogicExpression.rslib] at (-701.82, -354.86, 903.18) mm
        properties: Expression=FWD and not Error
    - NoErrorAllowREV [smart component, from Components\LogicExpression.rslib] at (-701.82, -354.86, 903.18) mm
        properties: Expression=REV and not Error
    - GraphicsShow [smart component, from Components\Show.rslib] at (-701.82, -354.86, 903.18) mm
        properties: Object=OnOffGfx
    - GraphicsHide [smart component, from Components\Hide.rslib] at (-701.82, -354.86, 903.18) mm
        properties: Object=OnOffGfx
    - GraphicsHideLogic [smart component, from Components\LogicExpression.rslib] at (-701.82, -354.86, 903.18) mm
        properties: Expression=not FWD and not REV
    - GraphicsObjects [graphiccomponentgroup] at (83.9, 149.37, 1003.18) mm, rotated rx 0 ry 0 rz -90 deg
      - OnOffGfx [graphiccomponentgroup] at (514.42, -850.96, -110.92) mm, rotated rx 0 ry 0 rz 90 deg
        - Part_5 [part] at (927.42, 264.29, 0) mm, rotated rx 0 ry 0 rz -90 deg, size 50 x 1493.5 x 100 mm
        - Part_6 [part] at (926.46, -134.61, 0) mm, rotated rx 0 ry 0 rz -90 deg, size 50 x 1492.5 x 100 mm
      - ConveyorSurface [part] at (-0.94, 65.23, -516.89) mm, rotated rx 0 ry 0 rz 180 deg, size 356.8 x 1451.8 x 107.9 mm
    - MotorFeedbackSignalLogic [smart component, from Components\LogicExpression.rslib] at (-701.82, -354.86, 903.18) mm
        properties: Expression=A AND NOT B
    - 1500x450x500 [graphiccomponentgroup] at (162.8, -49.34, 486.29) mm, rotated rx 0 ry 0 rz 180 deg
      - GeneratedPart [part] at (0, 0, 380) mm, size 1500 x 50 x 120 mm
      - GeneratedPart_2 [part] at (0, 400, 380) mm, size 1500 x 50 x 120 mm
      - GeneratedPart_3 [part] at (0, 50, 380) mm, size 50 x 350 x 120 mm
      - GeneratedPart_4 [part] at (1450, 50, 380) mm, size 50 x 350 x 120 mm
      - GeneratedPart_5 [part] at (150, 0, 72) mm
      - GeneratedPart_6 [part] at (150, 0, 72) mm
      - GeneratedPart_7 [part] at (150, 400, 72) mm
      - GeneratedPart_8 [part] at (125, 50, 460) mm, rotated rx -90 ry 0 rz 0 deg, size 80 x 79.7 x 350 mm
      - GeneratedPart_9 [part] at (162.5, -50, 0) mm
      - GeneratedPart_10 [part] at (162.5, -50, 0) mm
      - GeneratedPart_11 [part] at (162.5, 400, 0) mm
      - GeneratedPart_12 [part] at (125, 50, 460) mm, rotated rx -90 ry 0 rz 0 deg, size 80 x 79.7 x 350 mm
      - GeneratedPart_13 [part] at (250, 50, 460) mm, rotated rx -90 ry 0 rz 0 deg, size 80 x 79.7 x 350 mm
      - GeneratedPart_14 [part] at (375, 50, 460) mm, rotated rx -90 ry 0 rz 0 deg, size 80 x 79.7 x 350 mm
      - GeneratedPart_15 [part] at (500, 50, 460) mm, rotated rx -90 ry 0 rz 0 deg, size 80 x 79.7 x 350 mm
      - GeneratedPart_16 [part] at (625, 50, 460) mm, rotated rx -90 ry 0 rz 0 deg, size 80 x 79.7 x 350 mm
      - GeneratedPart_17 [part] at (750, 50, 460) mm, rotated rx -90 ry 0 rz 0 deg, size 80 x 79.7 x 350 mm
      - GeneratedPart_18 [part] at (875, 50, 460) mm, rotated rx -90 ry 0 rz 0 deg, size 80 x 79.7 x 350 mm
      - GeneratedPart_19 [part] at (1000, 50, 460) mm, rotated rx -90 ry 0 rz 0 deg, size 80 x 79.7 x 350 mm
      - GeneratedPart_20 [part] at (1125, 50, 460) mm, rotated rx -90 ry 0 rz 0 deg, size 80 x 79.7 x 350 mm
      - GeneratedPart_21 [part] at (1250, 50, 460) mm, rotated rx -90 ry 0 rz 0 deg, size 80 x 79.7 x 350 mm
      - GeneratedPart_22 [part] at (1375, 50, 460) mm, rotated rx -90 ry 0 rz 0 deg, size 80 x 79.7 x 350 mm
      - GeneratedPart_23 [part] at (200, 25, 12) mm
      - GeneratedPart_24 [part] at (200, 25, 12) mm
      - GeneratedPart_25 [part] at (200, 425, 12) mm
      - GeneratedPart_26 [part] at (1266.54, 400, 0) mm
      - GeneratedPart_27 [part] at (1254.04, 0, 72) mm
      - GeneratedPart_28 [part] at (1304.04, 25, 12) mm
      - GeneratedPart_29 [part] at (1266.54, -50, 0) mm
      - GeneratedPart_30 [part] at (1254.04, 400, 72) mm
      - GeneratedPart_31 [part] at (1304.04, 425, 12) mm
      - Part_3 [part] at (1105.7, 0.66, -486.29) mm, size 100 x 550 x 880 mm
      - Part_2 [part] at (0.3, 0.66, -486.29) mm, size 100 x 550 x 880 mm
    - SUB610_B1 [smart component] at (-13.16, -49.69, 870.13) mm, rotated rx 0 ry 0 rz 180 deg
        signals: DO SensorSignal
        connections:
          SensorRay.SensorOut -> ?.Active
          ?.Output -> SUB610_B1.SensorSignal
          SensorRay.SensorOut -> LogicGate.InputA
          GraphicSwitch_2.Output -> LogicGate_2.InputA
          LogicGate_2.Output -> LogicGate.InputB
          LogicGate.Output -> SUB610_B1.SensorSignal
      - SensorRay [smart component, from Components\LineSensor.rslib] at (24.04, 61.94, 174.13) mm
          properties: Start=[0 0 0]; End=[1.02087466601758E-07 0.23805885165687 4.04628539979468E-07]; Radius=0.01; SensedPart=(none); SensedPoint=[0 0 0]; Length=0.238058851657236; Tag=(none)
        - _sensorPart_ [part], size 20 x 238.1 x 20 mm
      - SensorMountWorking [part] at (0, 0, 0) mm, size 50 x 50 x 200 mm
      - GraphicSwitch_2 [smart component, from Components\GraphicSwitch.rslib] at (50, 0, 0) mm
          properties: PartHigh=SensorMountBroken; PartLow=SensorMountWorking
      - SensorMountBroken [part] at (0, 0, 0) mm, size 50 x 50 x 200 mm
      - LogicGate [smart component, from Components\LogicGate.rslib]
          properties: Operator=AND; Delay=0
      - LogicGate_2 [smart component, from Components\LogicGate.rslib]
          properties: Operator=NOT; Delay=0
  - SOP716 [smart component] at (3750, 10320, 100) mm, rotated rx 0 ry 0 rz 90 deg
      properties: ForwardSpeed=0.05; ReverseSpeed=-0.05; ConveyorSpeed=0; SpeedForward=0.7; Constant=1E-09; SpeedBackward=-0.6
      signals: DI MotorFWD, DI MotorREV, DO ConveyorError, DI ResetError, DO MotorFeedback, DO BoxSensor
      connections:
        SOP716.MotorFWD -> ?.Enabled
        SOP716.MotorREV -> ?.Enabled
        ?.Output -> ?.Enabled
        SOP716.MotorFWD -> ?.Execute
        SOP716.MotorREV -> ?.Execute
        SOP716.MotorFWD -> ?.A
        SOP716.MotorREV -> ?.B
        ?.Result -> ConveyorSurfaceBehaviour.SurfaceVelocity
        ?.Output -> ConveyorSurfaceBehaviour.SurfaceVelocity
        ?.Output -> ?.InputA
        ?.Output -> ?.InputB
        SOP716.MotorFWD -> ?.InputA
        SOP716.MotorFWD -> ?.InputA
        SOP716.MotorREV -> ?.InputB
        SOP716.MotorFWD -> ?.InputA
        SOP716.MotorFWD -> ?.A
        ?.Result -> ConveyorSurfaceBehaviour.SurfaceVelocity
        SOP716.MotorFWD -> ?.Set
        SOP716.MotorREV -> ?.Set
        SetIdleSpeed.Result -> SetIdleSpeedToConveyor.Execute
        SOP716.MotorFWD -> SetIdleSpeed.A
        SOP716.MotorREV -> SetIdleSpeed.B
        SOP716.MotorFWD -> SetMotorSafetyBreaker.FWD
        SOP716.MotorREV -> SetMotorSafetyBreaker.REV
        ErrorCheckAndBlockingMotorsAndErrorResetLogic.Output -> SetIdleSpeedToConveyor.Execute
        SOP716.ResetError -> ErrorCheckAndBlockingMotorsAndErrorResetLogic.Reset
        SOP716.MotorFWD -> NoErrorAllowFWD.FWD
        ErrorCheckAndBlockingMotorsAndErrorResetLogic.Output -> NoErrorAllowFWD.Error
        NoErrorAllowFWD.Result -> SetForwardSpeedToConveyor.Execute
        SOP716.MotorREV -> NoErrorAllowREV.REV
        ErrorCheckAndBlockingMotorsAndErrorResetLogic.Output -> NoErrorAllowREV.Error
        NoErrorAllowREV.Result -> SetBackwardSpeedToConveyor.Execute
        SetMotorSafetyBreaker.Result -> ErrorCheckAndBlockingMotorsAndErrorResetLogic.Set
        GraphicsHideLogic.Result -> GraphicsHide.Execute
        SOP716.MotorFWD -> GraphicsHideLogic.FWD
        SOP716.MotorREV -> GraphicsHideLogic.REV
        SOP716.MotorFWD -> MotorFeedbackSignalLogic.A
        SOP716.MotorREV -> MotorFeedbackSignalLogic.A
        ErrorCheckAndBlockingMotorsAndErrorResetLogic.Output -> MotorFeedbackSignalLogic.B
        MotorFeedbackSignalLogic.Result -> SOP716.MotorFeedback
        MotorFeedbackSignalLogic.Result -> GraphicsShow.Execute
        ErrorCheckAndBlockingMotorsAndErrorResetLogic.InvOutput -> SOP716.ConveyorError
        SUB610_B1.SensorSignal -> SOP716.BoxSensor
        ?.Result => ?.Count
        ?.Value => ConveyorSurfaceBehaviour.SurfaceVelocity
        ?.Value => ConveyorSurfaceBehaviour.SurfaceVelocity
        ?.Value => ConveyorSurfaceBehaviour.SurfaceVelocity
        ?.Value => ConveyorSurfaceBehaviour.SurfaceVelocity
        ?.Value => ConveyorSurfaceBehaviour.SurfaceVelocity
        ?.Value => ConveyorSurfaceBehaviour.SurfaceVelocity
        SetIdleSpeedToConveyor.Value => ConveyorSurfaceBehaviour.SurfaceVelocity
        SetForwardSpeedToConveyor.Value => ConveyorSurfaceBehaviour.SurfaceVelocity
        SetBackwardSpeedToConveyor.Value => ConveyorSurfaceBehaviour.SurfaceVelocity
        ?.Result => SetForwardSpeedToConveyor.Max
        ?.A => SetBackwardSpeedToConveyor.Min
        ?.Result => SetBackwardSpeedToConveyor.Max
        ?.A => SetForwardSpeedToConveyor.Min
        GraphicsShow.Object => GraphicsHide.Object
        ?.Object => ?.Object
    - ConveyorSurfaceBehaviour [smart component, from Components\PhysicsControl.rslib] at (-701.82, -354.86, 903.18) mm
        properties: Object=ConveyorSurface; Behavior=1; SurfaceVelocity=3.61908188723916E-14
    - SetIdleSpeedToConveyor [smart component, from Components\Random.rslib] at (-701.82, -354.86, 903.18) mm
        properties: Value=3.61908188723916E-14; Min=0; Max=1E-13
    - SetBackwardSpeedToConveyor [smart component, from Components\Random.rslib] at (-701.82, -354.86, 903.18) mm
        properties: Value=-0.69999999999997; Min=-0.7; Max=-0.6999999999999
    - SetForwardSpeedToConveyor [smart component, from Components\Random.rslib] at (-701.82, -354.86, 903.18) mm
        properties: Value=0.500000000072681; Min=0.5; Max=0.5000000001
    - SetIdleSpeed [smart component, from Components\LogicExpression.rslib] at (-701.82, -354.86, 903.18) mm
        properties: Expression=not A and not B
    - SetMotorSafetyBreaker [smart component, from Components\LogicExpression.rslib] at (-701.82, -354.86, 903.18) mm
        properties: Expression=FWD and REV
    - ErrorCheckAndBlockingMotorsAndErrorResetLogic [smart component, from Components\LogicSRLatch.rslib] at (-701.82, -354.86, 903.18) mm
    - NoErrorAllowFWD [smart component, from Components\LogicExpression.rslib] at (-701.82, -354.86, 903.18) mm
        properties: Expression=FWD and not Error
    - NoErrorAllowREV [smart component, from Components\LogicExpression.rslib] at (-701.82, -354.86, 903.18) mm
        properties: Expression=REV and not Error
    - GraphicsShow [smart component, from Components\Show.rslib] at (-701.82, -354.86, 903.18) mm
        properties: Object=OnOffGfx
    - GraphicsHide [smart component, from Components\Hide.rslib] at (-701.82, -354.86, 903.18) mm
        properties: Object=OnOffGfx
    - GraphicsHideLogic [smart component, from Components\LogicExpression.rslib] at (-701.82, -354.86, 903.18) mm
        properties: Expression=not FWD and not REV
    - GraphicsObjects [graphiccomponentgroup] at (83.9, 149.37, 1003.18) mm, rotated rx 0 ry 0 rz -90 deg
      - OnOffGfx [graphiccomponentgroup] at (514.42, -850.96, -110.92) mm, rotated rx 0 ry 0 rz 90 deg
        - Part_5 [part] at (927.42, 264.29, 0) mm, rotated rx 0 ry 0 rz -90 deg, size 50 x 1493.5 x 100 mm
        - Part_6 [part] at (926.46, -134.61, 0) mm, rotated rx 0 ry 0 rz -90 deg, size 50 x 1492.5 x 100 mm
      - ConveyorSurface [part] at (-0.94, 65.23, -516.89) mm, rotated rx 0 ry 0 rz 180 deg, size 356.8 x 1451.8 x 107.9 mm
    - MotorFeedbackSignalLogic [smart component, from Components\LogicExpression.rslib] at (-701.82, -354.86, 903.18) mm
        properties: Expression=A AND NOT B
    - 1500x450x500 [graphiccomponentgroup] at (162.8, -49.34, 486.29) mm, rotated rx 0 ry 0 rz 180 deg
      - GeneratedPart [part] at (0, 0, 380) mm, size 1500 x 50 x 120 mm
      - GeneratedPart_2 [part] at (0, 400, 380) mm, size 1500 x 50 x 120 mm
      - GeneratedPart_3 [part] at (0, 50, 380) mm, size 50 x 350 x 120 mm
      - GeneratedPart_4 [part] at (1450, 50, 380) mm, size 50 x 350 x 120 mm
      - GeneratedPart_5 [part] at (150, 0, 72) mm
      - GeneratedPart_6 [part] at (150, 0, 72) mm
      - GeneratedPart_7 [part] at (150, 400, 72) mm
      - GeneratedPart_8 [part] at (125, 50, 460) mm, rotated rx -90 ry 0 rz 0 deg, size 80 x 79.7 x 350 mm
      - GeneratedPart_9 [part] at (162.5, -50, 0) mm
      - GeneratedPart_10 [part] at (162.5, -50, 0) mm
      - GeneratedPart_11 [part] at (162.5, 400, 0) mm
      - GeneratedPart_12 [part] at (125, 50, 460) mm, rotated rx -90 ry 0 rz 0 deg, size 80 x 79.7 x 350 mm
      - GeneratedPart_13 [part] at (250, 50, 460) mm, rotated rx -90 ry 0 rz 0 deg, size 80 x 79.7 x 350 mm
      - GeneratedPart_14 [part] at (375, 50, 460) mm, rotated rx -90 ry 0 rz 0 deg, size 80 x 79.7 x 350 mm
      - GeneratedPart_15 [part] at (500, 50, 460) mm, rotated rx -90 ry 0 rz 0 deg, size 80 x 79.7 x 350 mm
      - GeneratedPart_16 [part] at (625, 50, 460) mm, rotated rx -90 ry 0 rz 0 deg, size 80 x 79.7 x 350 mm
      - GeneratedPart_17 [part] at (750, 50, 460) mm, rotated rx -90 ry 0 rz 0 deg, size 80 x 79.7 x 350 mm
      - GeneratedPart_18 [part] at (875, 50, 460) mm, rotated rx -90 ry 0 rz 0 deg, size 80 x 79.7 x 350 mm
      - GeneratedPart_19 [part] at (1000, 50, 460) mm, rotated rx -90 ry 0 rz 0 deg, size 80 x 79.7 x 350 mm
      - GeneratedPart_20 [part] at (1125, 50, 460) mm, rotated rx -90 ry 0 rz 0 deg, size 80 x 79.7 x 350 mm
      - GeneratedPart_21 [part] at (1250, 50, 460) mm, rotated rx -90 ry 0 rz 0 deg, size 80 x 79.7 x 350 mm
      - GeneratedPart_22 [part] at (1375, 50, 460) mm, rotated rx -90 ry 0 rz 0 deg, size 80 x 79.7 x 350 mm
      - GeneratedPart_23 [part] at (200, 25, 12) mm
      - GeneratedPart_24 [part] at (200, 25, 12) mm
      - GeneratedPart_25 [part] at (200, 425, 12) mm
      - GeneratedPart_26 [part] at (1266.54, 400, 0) mm
      - GeneratedPart_27 [part] at (1254.04, 0, 72) mm
      - GeneratedPart_28 [part] at (1304.04, 25, 12) mm
      - GeneratedPart_29 [part] at (1266.54, -50, 0) mm
      - GeneratedPart_30 [part] at (1254.04, 400, 72) mm
      - GeneratedPart_31 [part] at (1304.04, 425, 12) mm
      - Part_3 [part] at (1105.7, 0.66, -486.29) mm, size 100 x 550 x 880 mm
      - Part_2 [part] at (0.3, 0.66, -486.29) mm, size 100 x 550 x 880 mm
    - SUB610_B1 [smart component] at (-13.16, -49.69, 870.13) mm, rotated rx 0 ry 0 rz 180 deg
        signals: DO SensorSignal
        connections:
          SensorRay.SensorOut -> ?.Active
          ?.Output -> SUB610_B1.SensorSignal
          SensorRay.SensorOut -> LogicGate.InputA
          GraphicSwitch_2.Output -> LogicGate_2.InputA
          LogicGate_2.Output -> LogicGate.InputB
          LogicGate.Output -> SUB610_B1.SensorSignal
      - SensorRay [smart component, from Components\LineSensor.rslib] at (24.04, 61.94, 174.13) mm
          properties: Start=[0 0 0]; End=[1.02087466601758E-07 0.23805885165687 4.04628539979468E-07]; Radius=0.01; SensedPart=(none); SensedPoint=[0 0 0]; Length=0.238058851657236; Tag=(none)
        - _sensorPart_ [part], size 20 x 238.1 x 20 mm
      - SensorMountWorking [part] at (0, 0, 0) mm, size 50 x 50 x 200 mm
      - GraphicSwitch_2 [smart component, from Components\GraphicSwitch.rslib] at (50, 0, 0) mm
          properties: PartHigh=SensorMountBroken; PartLow=SensorMountWorking
      - SensorMountBroken [part] at (0, 0, 0) mm, size 50 x 50 x 200 mm
      - LogicGate [smart component, from Components\LogicGate.rslib]
          properties: Operator=AND; Delay=0
      - LogicGate_2 [smart component, from Components\LogicGate.rslib]
          properties: Operator=NOT; Delay=0
  - SOP713 [smart component] at (3750, 5820, 100) mm, rotated rx 0 ry 0 rz 90 deg
      properties: ForwardSpeed=0.05; ReverseSpeed=-0.05; ConveyorSpeed=0; SpeedForward=0.7; Constant=1E-09; SpeedBackward=-0.6
      signals: DI MotorFWD, DI MotorREV, DO ConveyorError, DI ResetError, DO MotorFeedback, DO BoxSensor, DO FrontUpSensor, DO RearUpSensor, DI FrontDown, DI FrontUp, DI RearDown, DI RearUp, DO FrontDownSensor, DO RareDownSensor
      connections:
        SOP713.MotorFWD -> ?.Enabled
        SOP713.MotorREV -> ?.Enabled
        ?.Output -> ?.Enabled
        SOP713.MotorFWD -> ?.Execute
        SOP713.MotorREV -> ?.Execute
        SOP713.MotorFWD -> ?.A
        SOP713.MotorREV -> ?.B
        ?.Result -> ConveyorSurfaceBehaviour.SurfaceVelocity
        ?.Output -> ConveyorSurfaceBehaviour.SurfaceVelocity
        ?.Output -> ?.InputA
        ?.Output -> ?.InputB
        SOP713.MotorFWD -> ?.InputA
        SOP713.MotorFWD -> ?.InputA
        SOP713.MotorREV -> ?.InputB
        SOP713.MotorFWD -> ?.InputA
        SOP713.MotorFWD -> ?.A
        ?.Result -> ConveyorSurfaceBehaviour.SurfaceVelocity
        SOP713.MotorFWD -> ?.Set
        SOP713.MotorREV -> ?.Set
        SetIdleSpeed.Result -> SetIdleSpeedToConveyor.Execute
        SOP713.MotorFWD -> SetIdleSpeed.A
        SOP713.MotorREV -> SetIdleSpeed.B
        SOP713.MotorFWD -> SetMotorSafetyBreaker.FWD
        SOP713.MotorREV -> SetMotorSafetyBreaker.REV
        ErrorCheckAndBlockingMotorsAndErrorResetLogic.Output -> SetIdleSpeedToConveyor.Execute
        SOP713.ResetError -> ErrorCheckAndBlockingMotorsAndErrorResetLogic.Reset
        SOP713.MotorFWD -> NoErrorAllowFWD.FWD
        ErrorCheckAndBlockingMotorsAndErrorResetLogic.Output -> NoErrorAllowFWD.Error
        NoErrorAllowFWD.Result -> SetForwardSpeedToConveyor.Execute
        SOP713.MotorREV -> NoErrorAllowREV.REV
        ErrorCheckAndBlockingMotorsAndErrorResetLogic.Output -> NoErrorAllowREV.Error
        NoErrorAllowREV.Result -> SetBackwardSpeedToConveyor.Execute
        SetMotorSafetyBreaker.Result -> ErrorCheckAndBlockingMotorsAndErrorResetLogic.Set
        GraphicsHideLogic.Result -> GraphicsHide.Execute
        SOP713.MotorFWD -> GraphicsHideLogic.FWD
        SOP713.MotorREV -> GraphicsHideLogic.REV
        SOP713.MotorFWD -> MotorFeedbackSignalLogic.A
        SOP713.MotorREV -> MotorFeedbackSignalLogic.A
        ErrorCheckAndBlockingMotorsAndErrorResetLogic.Output -> MotorFeedbackSignalLogic.B
        MotorFeedbackSignalLogic.Result -> SOP713.MotorFeedback
        MotorFeedbackSignalLogic.Result -> GraphicsShow.Execute
        ErrorCheckAndBlockingMotorsAndErrorResetLogic.InvOutput -> SOP713.ConveyorError
        SOP713.FrontDown -> SUB640 FrontClamp.ClampDown
        SOP713.FrontUp -> SUB640 FrontClamp.ClampUp
        SOP713.RearDown -> SUB640 RearClamp.ClampDown
        SOP713.RearUp -> SUB640 RearClamp.ClampUp
        SUB640_B1.SensorSignal -> SOP713.BoxSensor
        SUB640 FrontClamp.ClampUpPosition -> SOP713.FrontUpSensor
        SUB640 RearClamp.ClampUpPosition -> SOP713.RearUpSensor
        SUB640 RearClamp.ClampDownPosition -> SOP713.RareDownSensor
        SUB640 FrontClamp.ClampDownPosition -> SOP713.FrontDownSensor
        ?.Result => ?.Count
        ?.Value => ConveyorSurfaceBehaviour.SurfaceVelocity
        ?.Value => ConveyorSurfaceBehaviour.SurfaceVelocity
        ?.Value => ConveyorSurfaceBehaviour.SurfaceVelocity
        ?.Value => ConveyorSurfaceBehaviour.SurfaceVelocity
        ?.Value => ConveyorSurfaceBehaviour.SurfaceVelocity
        ?.Value => ConveyorSurfaceBehaviour.SurfaceVelocity
        SetIdleSpeedToConveyor.Value => ConveyorSurfaceBehaviour.SurfaceVelocity
        SetForwardSpeedToConveyor.Value => ConveyorSurfaceBehaviour.SurfaceVelocity
        SetBackwardSpeedToConveyor.Value => ConveyorSurfaceBehaviour.SurfaceVelocity
        ?.Result => SetForwardSpeedToConveyor.Max
        ?.A => SetBackwardSpeedToConveyor.Min
        ?.Result => SetBackwardSpeedToConveyor.Max
        ?.A => SetForwardSpeedToConveyor.Min
        GraphicsShow.Object => GraphicsHide.Object
        ?.Object => ?.Object
    - ConveyorSurfaceBehaviour [smart component, from Components\PhysicsControl.rslib] at (-701.82, -354.86, 903.18) mm
        properties: Object=ConveyorSurface; Behavior=1; SurfaceVelocity=6.57124071687983E-14
    - SetIdleSpeedToConveyor [smart component, from Components\Random.rslib] at (-701.82, -354.86, 903.18) mm
        properties: Value=6.57124071687983E-14; Min=0; Max=1E-13
    - SetBackwardSpeedToConveyor [smart component, from Components\Random.rslib] at (-701.82, -354.86, 903.18) mm
        properties: Value=-0.699999999999959; Min=-0.7; Max=-0.6999999999999
    - SetForwardSpeedToConveyor [smart component, from Components\Random.rslib] at (-701.82, -354.86, 903.18) mm
        properties: Value=0.500000000012043; Min=0.5; Max=0.5000000001
    - SetIdleSpeed [smart component, from Components\LogicExpression.rslib] at (-701.82, -354.86, 903.18) mm
        properties: Expression=not A and not B
    - SetMotorSafetyBreaker [smart component, from Components\LogicExpression.rslib] at (-701.82, -354.86, 903.18) mm
        properties: Expression=FWD and REV
    - ErrorCheckAndBlockingMotorsAndErrorResetLogic [smart component, from Components\LogicSRLatch.rslib] at (-701.82, -354.86, 903.18) mm
    - NoErrorAllowFWD [smart component, from Components\LogicExpression.rslib] at (-701.82, -354.86, 903.18) mm
        properties: Expression=FWD and not Error
    - NoErrorAllowREV [smart component, from Components\LogicExpression.rslib] at (-701.82, -354.86, 903.18) mm
        properties: Expression=REV and not Error
    - GraphicsShow [smart component, from Components\Show.rslib] at (-701.82, -354.86, 903.18) mm
        properties: Object=OnOffGfx
    - GraphicsHide [smart component, from Components\Hide.rslib] at (-701.82, -354.86, 903.18) mm
        properties: Object=OnOffGfx
    - GraphicsHideLogic [smart component, from Components\LogicExpression.rslib] at (-701.82, -354.86, 903.18) mm
        properties: Expression=not FWD and not REV
    - GraphicsObjects [graphiccomponentgroup] at (83.9, 149.37, 1003.18) mm, rotated rx 0 ry 0 rz -90 deg
      - OnOffGfx [graphiccomponentgroup] at (514.42, -850.96, -110.92) mm, rotated rx 0 ry 0 rz 90 deg
        - Part_5 [part] at (927.42, 264.29, 0) mm, rotated rx 0 ry 0 rz -90 deg, size 50 x 1493.5 x 100 mm
        - Part_6 [part] at (926.46, -134.61, 0) mm, rotated rx 0 ry 0 rz -90 deg, size 50 x 1492.5 x 100 mm
      - ConveyorSurface [part] at (-0.94, 65.23, -516.89) mm, rotated rx 0 ry 0 rz 180 deg, size 356.8 x 1451.8 x 107.9 mm
    - MotorFeedbackSignalLogic [smart component, from Components\LogicExpression.rslib] at (-701.82, -354.86, 903.18) mm
        properties: Expression=A AND NOT B
    - 1500x450x500 [graphiccomponentgroup] at (162.8, -49.34, 486.29) mm, rotated rx 0 ry 0 rz 180 deg
      - GeneratedPart [part] at (0, 0, 380) mm, size 1500 x 50 x 120 mm
      - GeneratedPart_2 [part] at (0, 400, 380) mm, size 1500 x 50 x 120 mm
      - GeneratedPart_3 [part] at (0, 50, 380) mm, size 50 x 350 x 120 mm
      - GeneratedPart_4 [part] at (1450, 50, 380) mm, size 50 x 350 x 120 mm
      - GeneratedPart_5 [part] at (150, 0, 72) mm
      - GeneratedPart_6 [part] at (150, 0, 72) mm
      - GeneratedPart_7 [part] at (150, 400, 72) mm
      - GeneratedPart_8 [part] at (125, 50, 460) mm, rotated rx -90 ry 0 rz 0 deg, size 80 x 79.7 x 350 mm
      - GeneratedPart_9 [part] at (162.5, -50, 0) mm
      - GeneratedPart_10 [part] at (162.5, -50, 0) mm
      - GeneratedPart_11 [part] at (162.5, 400, 0) mm
      - GeneratedPart_12 [part] at (125, 50, 460) mm, rotated rx -90 ry 0 rz 0 deg, size 80 x 79.7 x 350 mm
      - GeneratedPart_13 [part] at (250, 50, 460) mm, rotated rx -90 ry 0 rz 0 deg, size 80 x 79.7 x 350 mm
      - GeneratedPart_14 [part] at (375, 50, 460) mm, rotated rx -90 ry 0 rz 0 deg, size 80 x 79.7 x 350 mm
      - GeneratedPart_15 [part] at (500, 50, 460) mm, rotated rx -90 ry 0 rz 0 deg, size 80 x 79.7 x 350 mm
      - GeneratedPart_16 [part] at (625, 50, 460) mm, rotated rx -90 ry 0 rz 0 deg, size 80 x 79.7 x 350 mm
      - GeneratedPart_17 [part] at (750, 50, 460) mm, rotated rx -90 ry 0 rz 0 deg, size 80 x 79.7 x 350 mm
      - GeneratedPart_18 [part] at (875, 50, 460) mm, rotated rx -90 ry 0 rz 0 deg, size 80 x 79.7 x 350 mm
      - GeneratedPart_19 [part] at (1000, 50, 460) mm, rotated rx -90 ry 0 rz 0 deg, size 80 x 79.7 x 350 mm
      - GeneratedPart_20 [part] at (1125, 50, 460) mm, rotated rx -90 ry 0 rz 0 deg, size 80 x 79.7 x 350 mm
      - GeneratedPart_21 [part] at (1250, 50, 460) mm, rotated rx -90 ry 0 rz 0 deg, size 80 x 79.7 x 350 mm
      - GeneratedPart_22 [part] at (1375, 50, 460) mm, rotated rx -90 ry 0 rz 0 deg, size 80 x 79.7 x 350 mm
      - GeneratedPart_23 [part] at (200, 25, 12) mm
      - GeneratedPart_24 [part] at (200, 25, 12) mm
      - GeneratedPart_25 [part] at (200, 425, 12) mm
      - GeneratedPart_26 [part] at (1266.54, 400, 0) mm
      - GeneratedPart_27 [part] at (1254.04, 0, 72) mm
      - GeneratedPart_28 [part] at (1304.04, 25, 12) mm
      - GeneratedPart_29 [part] at (1266.54, -50, 0) mm
      - GeneratedPart_30 [part] at (1254.04, 400, 72) mm
      - GeneratedPart_31 [part] at (1304.04, 425, 12) mm
      - Part_3 [part] at (1105.7, 0.66, -486.29) mm, size 100 x 550 x 880 mm
      - Part_2 [part] at (0.3, 0.66, -486.29) mm, size 100 x 550 x 880 mm
    - SUB640 FrontClamp [smart component] at (-13.06, -370.35, 892.01) mm, rotated rx 0 ry 0 rz 90 deg
        signals: DI ClampUp, DI ClampDown, DO ClampUpPosition, DO ClampDownPosition
        connections:
          SUB640 FrontClamp.ClampUp -> LogicExpression.A
          BottomPosSensor.SensorOut -> LogicExpression.B
          LogicExpression.Result -> LinearMoveUp.Execute
          SUB640 FrontClamp.ClampDown -> LogicExpression_2.A
          BottomPosSensor.SensorOut -> LogicExpression_2.B
          LogicExpression_2.Result -> LinearMoveDown.Execute
          LinearMoveUp.Executed -> LogicSRLatch.Set
          LogicSRLatch.Output -> SUB640 FrontClamp.ClampUpPosition
          LinearMoveDown.Executed -> ?.Set
          ?.Output -> SUB640 FrontClamp.ClampDownPosition
          LinearMoveDown.Executing -> LogicSRLatch.Reset
          LinearMoveUp.Executing -> ?.Reset
          BottomPosSensor.SensorOut -> SUB640 FrontClamp.ClampDownPosition
      - Clamp3D [part] at (0, 0, 100) mm, size 200 x 25 x 70 mm
      - BottomPosSensor [smart component, from Components\LineSensor.rslib] at (18.37, 10.91, 93.4) mm
          properties: Start=[-5.44677247749092E-09 -9.84894448774476E-08 -0.0999997155196143]; End=[-5.44677247749092E-09 -9.84894448774476E-08 -0.0899997155196144]; Radius=0.02; SensedPart=(none); SensedPoint=[0 0 0]; Length=0.0099999999999999; Tag=(none)
        - _sensorPart_ [part], size 40 x 40 x 10 mm
      - LinearMoveUp [smart component, from Components\LinearMover2.rslib]
          properties: Object=Clamp3D; Direction=[0 0 0.1]; Distance=0.1; Duration=1; Reference=Global; ReferenceObject=(none)
      - LinearMoveDown [smart component, from Components\LinearMover2.rslib]
          properties: Object=Clamp3D; Direction=[0 0 -0.1]; Distance=0.1; Duration=1; Reference=Global; ReferenceObject=(none)
      - LogicExpression [smart component, from Components\LogicExpression.rslib]
          properties: Expression=A AND B
      - LogicExpression_2 [smart component, from Components\LogicExpression.rslib]
          properties: Expression=A AND NOT B
      - LogicSRLatch [smart component, from Components\LogicSRLatch.rslib]
    - SUB640 RearClamp [smart component] at (-1013.6, -370.35, 892.01) mm, rotated rx 0 ry 0 rz 90 deg
        signals: DI ClampUp, DI ClampDown, DO ClampUpPosition, DO ClampDownPosition
        connections:
          SUB640 RearClamp.ClampUp -> LogicExpression.A
          BottomPosSensor.SensorOut -> LogicExpression.B
          LogicExpression.Result -> LinearMoveUp.Execute
          SUB640 RearClamp.ClampDown -> LogicExpression_2.A
          BottomPosSensor.SensorOut -> LogicExpression_2.B
          LogicExpression_2.Result -> LinearMoveDown.Execute
          LinearMoveUp.Executed -> LogicSRLatch.Set
          LogicSRLatch.Output -> SUB640 RearClamp.ClampUpPosition
          LinearMoveDown.Executed -> ?.Set
          ?.Output -> SUB640 RearClamp.ClampDownPosition
          LinearMoveDown.Executing -> LogicSRLatch.Reset
          LinearMoveUp.Executing -> ?.Reset
          BottomPosSensor.SensorOut -> SUB640 RearClamp.ClampDownPosition
      - Clamp3D [part] at (0, 0, 100) mm, size 200 x 25 x 70 mm
      - BottomPosSensor [smart component, from Components\LineSensor.rslib] at (18.37, 10.91, 93.4) mm
          properties: Start=[-5.44677247749092E-09 -9.84894448774476E-08 -0.0999997155196143]; End=[-5.44677247749092E-09 -9.84894448774476E-08 -0.0899997155196144]; Radius=0.02; SensedPart=(none); SensedPoint=[0 0 0]; Length=0.0099999999999999; Tag=(none)
        - _sensorPart_ [part], size 40 x 40 x 10 mm
      - LinearMoveUp [smart component, from Components\LinearMover2.rslib]
          properties: Object=Clamp3D; Direction=[0 0 0.1]; Distance=0.1; Duration=1; Reference=Global; ReferenceObject=(none)
      - LinearMoveDown [smart component, from Components\LinearMover2.rslib]
          properties: Object=Clamp3D; Direction=[0 0 -0.1]; Distance=0.1; Duration=1; Reference=Global; ReferenceObject=(none)
      - LogicExpression [smart component, from Components\LogicExpression.rslib]
          properties: Expression=A AND B
      - LogicExpression_2 [smart component, from Components\LogicExpression.rslib]
          properties: Expression=A AND NOT B
      - LogicSRLatch [smart component, from Components\LogicSRLatch.rslib]
    - SUB640_B1 [smart component] at (-66.51, -49.69, 870.13) mm, rotated rx 0 ry 0 rz 180 deg
        signals: DO SensorSignal
        connections:
          SensorRay.SensorOut -> ?.Active
          ?.Output -> SUB640_B1.SensorSignal
          SensorRay.SensorOut -> LogicGate.InputA
          GraphicSwitch_2.Output -> LogicGate_2.InputA
          LogicGate_2.Output -> LogicGate.InputB
          LogicGate.Output -> SUB640_B1.SensorSignal
      - SensorRay [smart component, from Components\LineSensor.rslib] at (24.04, 61.94, 174.13) mm
          properties: Start=[0 0 0]; End=[1.02087466601758E-07 0.23805885165687 4.04628539979468E-07]; Radius=0.01; SensedPart=(none); SensedPoint=[0 0 0]; Length=0.238058851657236; Tag=(none)
        - _sensorPart_ [part], size 20 x 238.1 x 20 mm
      - SensorMountWorking [part] at (0, 0, 0) mm, size 50 x 50 x 200 mm
      - GraphicSwitch_2 [smart component, from Components\GraphicSwitch.rslib] at (50, 0, 0) mm
          properties: PartHigh=SensorMountBroken; PartLow=SensorMountWorking
      - SensorMountBroken [part] at (0, 0, 0) mm, size 50 x 50 x 200 mm
      - LogicGate [smart component, from Components\LogicGate.rslib]
          properties: Operator=AND; Delay=0
      - LogicGate_2 [smart component, from Components\LogicGate.rslib]
          properties: Operator=NOT; Delay=0
  - Fences [graphiccomponentgroup]
    - Light Curtains [graphiccomponentgroup]
      - Light Curtain 4 [graphiccomponentgroup] at (7449.67, 2607.38, 100) mm, rotated rx 0 ry 0 rz 180 deg
        - Segment 1 [part], size 184 x 44 x 2000 mm
        - Segment 2 [part], size 184 x 2022 x 2000 mm
        - North Fence [graphiccomponentgroup] at (7449.67, 2607.38, -100) mm, rotated rx 0 ry 0 rz 180 deg
          - Segment 1 [part], size 184 x 44 x 2000 mm
          - Segment 2 [part], size 184 x 1500 x 2000 mm
          - Segment 3 [part], size 184 x 1522 x 2000 mm
          - Segment 4 [part], size 184 x 1522 x 2000 mm
          - Segment 5 [part], size 184 x 1522 x 2000 mm
          - Segment 6 [part], size 184 x 1522 x 2000 mm
          - Segment 7 [part], size 184 x 1522 x 2000 mm
          - Segment 8 [part], size 184 x 1522 x 2000 mm
          - Segment 9 [part], size 184 x 1500 x 2000 mm
      - Light Curtain 3 [graphiccomponentgroup] at (7448.79, 2609.72, 100) mm, rotated rx 0 ry 0 rz 180 deg
        - Segment 1 [part], size 44 x 184 x 2000 mm
        - Segment 2 [part] at (0, 0, 30) mm, size 2022 x 184 x 2000 mm
        - Segment 2 [part], size 422 x 184 x 2000 mm
      - Light Curtain 1 [graphiccomponentgroup] at (7446.09, 9609.65, 100) mm, rotated rx 0 ry 0 rz 180 deg
        - Segment 1 [part], size 44 x 184 x 2000 mm
        - Segment 2 [part], size 2022 x 184 x 2000 mm
        - Segment 2 [part], size 342 x 184 x 2000 mm
      - Light Curtain 2 [graphiccomponentgroup] at (7446.09, 7770.23, 100) mm, rotated rx 0 ry 0 rz 180 deg
        - Segment 1 [part], size 44 x 184 x 2000 mm
        - Segment 2 [part], size 2022 x 184 x 2000 mm
        - Segment 2 [part], size 342 x 184 x 2000 mm
    - South Fences [graphiccomponentgroup]
      - South Fence [graphiccomponentgroup] at (4782.42, 9612.49, 100) mm
        - Segment 2 [part] at (378.54, -41.71, 0) mm, size 184 x 882 x 2000 mm
      - South Fence 2 [graphiccomponentgroup] at (7446.26, 2608.99, 100) mm
        - Segment 1 [part], size 184 x 44 x 2000 mm
        - Segment 2 [part], size 184 x 1743 x 2000 mm
        - Segment 3 [part], size 184 x 1743 x 2000 mm
        - Segment 4 [part], size 184 x 1743 x 2000 mm
      - South Fence 3 [graphiccomponentgroup] at (5047.64, 610.05, 100) mm
        - Segment 1 [part], size 184 x 44 x 2000 mm
        - Segment 2 [part], size 184 x 2022 x 2000 mm
      - South Fence 5 [graphiccomponentgroup] at (5126.72, 7770.8, 100) mm
        - Segment 1 [part], size 184 x 44 x 2000 mm
        - Segment 2 [part], size 184 x 1863 x 2000 mm
      - South Fence 6 [graphiccomponentgroup] at (7434.45, 7770.31, 100) mm
        - Segment 1 [part], size 184 x 44 x 2000 mm
        - Segment 2 [part], size 184 x 1862 x 2000 mm
      - South Fence 8 [graphiccomponentgroup] at (7444.63, 22.88, 100) mm
        - Segment 1 [part], size 184 x 44 x 2000 mm
        - Segment 2 [part], size 184 x 607 x 2000 mm
      - South Fence 4 [graphiccomponentgroup] at (7449.38, 608.38, 100) mm, rotated rx 0 ry 0 rz 180 deg
        - Segment 1 [part], size 44 x 184 x 2000 mm
        - Segment 2 [part], size 2022 x 184 x 2000 mm
        - Segment 2 [part], size 422 x 184 x 2000 mm
      - South Fence 1 [graphiccomponentgroup] at (5160.63, 11231.82, 100) mm, rotated rx 0 ry 0 rz 180 deg
        - Segment 1 [part], size 44 x 184 x 2000 mm
        - Segment 2 [part], size 722 x 184 x 2000 mm
      - South Fence 9 [graphiccomponentgroup] at (4460.44, 11232.2, 100) mm, rotated rx 0 ry 0 rz 90 deg
        - Segment 1 [part], size 44 x 184 x 2000 mm
        - Segment 2 [part], size 782 x 184 x 2000 mm
  - IRC5_Dual-Cabinet [part, from %ABB.RobotStudio.Models.IRC5%\IRC5_Dual-Cabinet.rslib] at (5057.63, 11621.32, 200) mm, rotated rx 90 ry 0 rz 90 deg
  - HMI [graphiccomponentgroup, from Components\HMI.rslib] at (5433.14, 10003.79, 100) mm, rotated rx 0 ry 0 rz 90 deg
    - Foot [part, from Components\HMI.rslib] at (-7.27, 0.81, 0) mm, rotated rx 0 ry 0 rz 120 deg
    - Cylinder [part, from Components\HMI.rslib] at (3371.31, -375.11, 491.02) mm
    - Top Box [part, from Components\HMI.rslib] at (-254.89, -119.14, 1049.49) mm
  - SUB700LightBeacon [smart component, from Components\Light Beacon Large v0.2.rslib] at (5363.67, 9937.88, 2331) mm
      connections:
        SUB700LightBeacon.RedLight -> Red.Input
        SUB700LightBeacon.AmberLight -> Amber.Input
        SUB700LightBeacon.GreenLight -> Green.Input
        SUB700LightBeacon.BlueLight -> Blue.Input
    - LRedON [part, from Components\Light Beacon Large v0.2.rslib] at (0, 0, -110.52) mm
    - LAmberOFF [part, from Components\Light Beacon Large v0.2.rslib] at (0, 0, -207.79) mm
    - LAmberON [part, from Components\Light Beacon Large v0.2.rslib] at (0, 0, -207.79) mm
    - LBlueOFF [part, from Components\Light Beacon Large v0.2.rslib] at (0, 0, -403.44) mm
    - LBlueON [part, from Components\Light Beacon Large v0.2.rslib] at (0, 0, -403.44) mm
    - LGreenOFF [part, from Components\Light Beacon Large v0.2.rslib] at (0, 0, -307.9) mm
    - LGreenON [part, from Components\Light Beacon Large v0.2.rslib] at (0, 0, -307.9) mm
    - LPla5te [part, from Components\Light Beacon Large v0.2.rslib] at (0, 0, -20) mm
    - LPlate1 [part, from Components\Light Beacon Large v0.2.rslib] at (0, 0, -403.44) mm
    - LPlate2 [part, from Components\Light Beacon Large v0.2.rslib] at (0, 0, -314.18) mm
    - LPlate3 [part, from Components\Light Beacon Large v0.2.rslib] at (0, 0, -217.7) mm
    - LPlate4 [part, from Components\Light Beacon Large v0.2.rslib] at (0, 0, -120.06) mm
    - LRedOFF [part, from Components\Light Beacon Large v0.2.rslib] at (0, 0, -110.52) mm
    - Red [smart component, from Components\GraphicSwitch.rslib] at (1518.63, -1680.27, -2058.09) mm
        properties: PartHigh=LRedON; PartLow=LRedOFF
    - Amber [smart component, from Components\GraphicSwitch.rslib] at (1518.63, -1680.27, -2058.09) mm
        properties: PartHigh=LAmberON; PartLow=LAmberOFF
    - Green [smart component, from Components\GraphicSwitch.rslib] at (1518.63, -1680.27, -2058.09) mm
        properties: PartHigh=LGreenON; PartLow=LGreenOFF
    - Blue [smart component, from Components\GraphicSwitch.rslib] at (1518.63, -1680.27, -2058.09) mm
        properties: PartHigh=LBlueON; PartLow=LBlueOFF
    - Stand [part, from Components\Light Beacon Large v0.2.rslib] at (3.48, 0.46, -691.48) mm
  - HMI 1 [part], size 300 x 90 x 50 mm
  - HMI 2 [part] at (0, 6953.06, 0) mm, size 300 x 90 x 50 mm
  - SUB700LightBeacon 2 [smart component, from Components\Light Beacon Large v0.2.rslib] at (7442.18, 9581.01, 2809.9) mm
      connections:
        SUB700LightBeacon 2.RedLight -> Red.Input
        SUB700LightBeacon 2.AmberLight -> Amber.Input
        SUB700LightBeacon 2.GreenLight -> Green.Input
        SUB700LightBeacon 2.BlueLight -> Blue.Input
    - LRedON [part, from Components\Light Beacon Large v0.2.rslib] at (0, 0, -110.52) mm
    - LAmberOFF [part, from Components\Light Beacon Large v0.2.rslib] at (0, 0, -207.79) mm
    - LAmberON [part, from Components\Light Beacon Large v0.2.rslib] at (0, 0, -207.79) mm
    - LBlueOFF [part, from Components\Light Beacon Large v0.2.rslib] at (0, 0, -403.44) mm
    - LBlueON [part, from Components\Light Beacon Large v0.2.rslib] at (0, 0, -403.44) mm
    - LGreenOFF [part, from Components\Light Beacon Large v0.2.rslib] at (0, 0, -307.9) mm
    - LGreenON [part, from Components\Light Beacon Large v0.2.rslib] at (0, 0, -307.9) mm
    - LPla5te [part, from Components\Light Beacon Large v0.2.rslib] at (0, 0, -20) mm
    - LPlate1 [part, from Components\Light Beacon Large v0.2.rslib] at (0, 0, -403.44) mm
    - LPlate2 [part, from Components\Light Beacon Large v0.2.rslib] at (0, 0, -314.18) mm
    - LPlate3 [part, from Components\Light Beacon Large v0.2.rslib] at (0, 0, -217.7) mm
    - LPlate4 [part, from Components\Light Beacon Large v0.2.rslib] at (0, 0, -120.06) mm
    - LRedOFF [part, from Components\Light Beacon Large v0.2.rslib] at (0, 0, -110.52) mm
    - Red [smart component, from Components\GraphicSwitch.rslib] at (1518.63, -1680.27, -2058.09) mm
        properties: PartHigh=LRedON; PartLow=LRedOFF
    - Amber [smart component, from Components\GraphicSwitch.rslib] at (1518.63, -1680.27, -2058.09) mm
        properties: PartHigh=LAmberON; PartLow=LAmberOFF
    - Green [smart component, from Components\GraphicSwitch.rslib] at (1518.63, -1680.27, -2058.09) mm
        properties: PartHigh=LGreenON; PartLow=LGreenOFF
    - Blue [smart component, from Components\GraphicSwitch.rslib] at (1518.63, -1680.27, -2058.09) mm
        properties: PartHigh=LBlueON; PartLow=LBlueOFF
    - Stand [part, from Components\Light Beacon Large v0.2.rslib] at (3.48, 0.46, -691.48) mm
  - SUB700LightBeacon 3 [smart component, from Components\Light Beacon Large v0.2.rslib] at (7445.66, 2632.24, 2861.86) mm
      connections:
        SUB700LightBeacon 3.RedLight -> Red.Input
        SUB700LightBeacon 3.AmberLight -> Amber.Input
        SUB700LightBeacon 3.GreenLight -> Green.Input
        SUB700LightBeacon 3.BlueLight -> Blue.Input
    - LRedON [part, from Components\Light Beacon Large v0.2.rslib] at (0, 0, -110.52) mm
    - LAmberOFF [part, from Components\Light Beacon Large v0.2.rslib] at (0, 0, -207.79) mm
    - LAmberON [part, from Components\Light Beacon Large v0.2.rslib] at (0, 0, -207.79) mm
    - LBlueOFF [part, from Components\Light Beacon Large v0.2.rslib] at (0, 0, -403.44) mm
    - LBlueON [part, from Components\Light Beacon Large v0.2.rslib] at (0, 0, -403.44) mm
    - LGreenOFF [part, from Components\Light Beacon Large v0.2.rslib] at (0, 0, -307.9) mm
    - LGreenON [part, from Components\Light Beacon Large v0.2.rslib] at (0, 0, -307.9) mm
    - LPla5te [part, from Components\Light Beacon Large v0.2.rslib] at (0, 0, -20) mm
    - LPlate1 [part, from Components\Light Beacon Large v0.2.rslib] at (0, 0, -403.44) mm
    - LPlate2 [part, from Components\Light Beacon Large v0.2.rslib] at (0, 0, -314.18) mm
    - LPlate3 [part, from Components\Light Beacon Large v0.2.rslib] at (0, 0, -217.7) mm
    - LPlate4 [part, from Components\Light Beacon Large v0.2.rslib] at (0, 0, -120.06) mm
    - LRedOFF [part, from Components\Light Beacon Large v0.2.rslib] at (0, 0, -110.52) mm
    - Red [smart component, from Components\GraphicSwitch.rslib] at (1518.63, -1680.27, -2058.09) mm
        properties: PartHigh=LRedON; PartLow=LRedOFF
    - Amber [smart component, from Components\GraphicSwitch.rslib] at (1518.63, -1680.27, -2058.09) mm
        properties: PartHigh=LAmberON; PartLow=LAmberOFF
    - Green [smart component, from Components\GraphicSwitch.rslib] at (1518.63, -1680.27, -2058.09) mm
        properties: PartHigh=LGreenON; PartLow=LGreenOFF
    - Blue [smart component, from Components\GraphicSwitch.rslib] at (1518.63, -1680.27, -2058.09) mm
        properties: PartHigh=LBlueON; PartLow=LBlueOFF
    - Stand [part, from Components\Light Beacon Large v0.2.rslib] at (3.48, 0.46, -691.48) mm
  - OpcUaClient [smart component, from Components\OpcUaClient.rslib]
      properties: Status=Conectado; ServerAddress=opc.tcp://localhost:4840; UseSecurity=false; AutoConnect=true; Blocking=false; Authentication=0; SignalConfiguration=NamespaceUri;IdentifierType;Identifier;ReadWrite;Signal;SignalType;Controller;Device
CODESYSSPV3/3S/IecVarAccess;String;|var|CODESYS Control Win V3 x64.Application.IOs.SOP700_NS1;Write;SOP700_NS1;Digital;;
CODESYSSPV3/3S/IecVarAccess;String;|var|CODESYS Control Win V3 x64.Application.IOs.SOP720_HMI_NS1;Write;SOP720_HMI_NS1;Digital;;
CODESYSSPV3/3S/IecVarAccess;String;|var|CODESYS Control Win V3 x64.Application.IOs.SOP723_HMI_NS1;Write;SOP723_HMI_NS1;Digital;;
CODESYSSPV3/3S/IecVarAccess;String;|var|CODESYS Control Win V3 x64.Application.IOs.SOP750_FQ1;Write;SOP750_FQ1;Digital;;
CODESYSSPV3/3S/IecVarAccess;String;|var|CODESYS Control Win V3 x64.Application.IOs.SOP751_FQ1;Write;SOP751_FQ1;Digital;;
CODESYSSPV3/3S/IecVarAccess;String;|var|CODESYS Control Win V3 x64.Application.IOs.SOP751_F10;Write;SOP751_F10;Digital;;
CODESYSSPV3/3S/IecVarAccess;String;|var|CODESYS Control Win V3 x64.Application.IOs.SOP751_F11;Write;SOP751_F11;Digital;;
CODESYSSPV3/3S/IecVarAccess;String;|var|CODESYS Control Win V3 x64.Application.IOs.SOP751_F12;Write;SOP751_F12;Digital;;
CODESYSSPV3/3S/IecVarAccess;String;|var|CODESYS Control Win V3 x64.Application.IOs.SOP751_F13;Write;SOP751_F13;Digital;;
CODESYSSPV3/3S/IecVarAccess;String;|var|CODESYS Control Win V3 x64.Application.IOs.SOP750_K1;Write;SOP750_K1;Digital;;
CODESYSSPV3/3S/IecVarAccess;String;|var|CODESYS Control Win V3 x64.Application.IOs.SOP750_B1;Write;SOP750_B1;Digital;;
CODESYSSPV3/3S/IecVarAccess;String;|var|CODESYS Control Win V3 x64.Application.IOs.SOP750_K8;Write;SOP750_K8;Digital;;
CODESYSSPV3/3S/IecVarAccess;String;|var|CODESYS Control Win V3 x64.Application.IOs.SOP750_B2;Write;SOP750_B2;Digital;;
CODESYSSPV3/3S/IecVarAccess;String;|var|CODESYS Control Win V3 x64.Application.IOs.SOP750_B3;Write;SOP750_B3;Digital;;
CODESYSSPV3/3S/IecVarAccess;String;|var|CODESYS Control Win V3 x64.Application.IOs.SOP740_RobotReady;Write;SOP740_RobotReady;Digital;;
CODESYSSPV3/3S/IecVarAccess;String;|var|CODESYS Control Win V3 x64.Application.IOs.SOP740_ProductPlaced;Write;SOP740_ProductPlaced;Digital;;
CODESYSSPV3/3S/IecVarAccess;String;|var|CODESYS Control Win V3 x64.Application.IOs.SOP710_FQ1;Write;SOP710_FQ1;Digital;;
CODESYSSPV3/3S/IecVarAccess;String;|var|CODESYS Control Win V3 x64.Application.IOs.SOP710_B1;Write;SOP710_B1;Digital;;
CODESYSSPV3/3S/IecVarAccess;String;|var|CODESYS Control Win V3 x64.Application.IOs.SOP711_FQ1;Write;SOP711_FQ1;Digital;;
CODESYSSPV3/3S/IecVarAccess;String;|var|CODESYS Control Win V3 x64.Application.IOs.SOP711_B1;Write;SOP711_B1;Digital;;
CODESYSSPV3/3S/IecVarAccess;String;|var|CODESYS Control Win V3 x64.Application.IOs.SOP712_FQ1;Write;SOP712_FQ1;Digital;;
CODESYSSPV3/3S/IecVarAccess;String;|var|CODESYS Control Win V3 x64.Application.IOs.SOP712_B1;Write;SOP712_B1;Digital;;
CODESYSSPV3/3S/IecVarAccess;String;|var|CODESYS Control Win V3 x64.Application.IOs.SOP713_FQ1;Write;SOP713_FQ1;Digital;;
CODESYSSPV3/3S/IecVarAccess;String;|var|CODESYS Control Win V3 x64.Application.IOs.SOP713_B1;Write;SOP713_B1;Digital;;
CODESYSSPV3/3S/IecVarAccess;String;|var|CODESYS Control Win V3 x64.Application.IOs.SOP713_B2;Write;SOP713_B2;Digital;;
CODESYSSPV3/3S/IecVarAccess;String;|var|CODESYS Control Win V3 x64.Application.IOs.SOP713_B3;Write;SOP713_B3;Digital;;
CODESYSSPV3/3S/IecVarAccess;String;|var|CODESYS Control Win V3 x64.Application.IOs.SOP714_FQ1;Write;SOP714_FQ1;Digital;;
CODESYSSPV3/3S/IecVarAccess;String;|var|CODESYS Control Win V3 x64.Application.IOs.SOP714_B1;Write;SOP714_B1;Digital;;
CODESYSSPV3/3S/IecVarAccess;String;|var|CODESYS Control Win V3 x64.Application.IOs.SOP715_FQ1;Write;SOP715_FQ1;Digital;;
CODESYSSPV3/3S/IecVarAccess;String;|var|CODESYS Control Win V3 x64.Application.IOs.SOP715_B1;Write;SOP715_B1;Digital;;
CODESYSSPV3/3S/IecVarAccess;String;|var|CODESYS Control Win V3 x64.Application.IOs.SOP716_FQ1;Write;SOP716_FQ1;Digital;;
CODESYSSPV3/3S/IecVarAccess;String;|var|CODESYS Control Win V3 x64.Application.IOs.SOP716_B1;Write;SOP716_B1;Digital;;
CODESYSSPV3/3S/IecVarAccess;String;|var|CODESYS Control Win V3 x64.Application.IOs.SOP717_FQ1;Write;SOP717_FQ1;Digital;;
CODESYSSPV3/3S/IecVarAccess;String;|var|CODESYS Control Win V3 x64.Application.IOs.SOP717_B1;Write;SOP717_B1;Digital;;
CODESYSSPV3/3S/IecVarAccess;String;|var|CODESYS Control Win V3 x64.Application.IOs.SOP720_FQ1;Write;SOP720_FQ1;Digital;;
CODESYSSPV3/3S/IecVarAccess;String;|var|CODESYS Control Win V3 x64.Application.IOs.SOP720_B1;Write;SOP720_B1;Digital;;
CODESYSSPV3/3S/IecVarAccess;String;|var|CODESYS Control Win V3 x64.Application.IOs.SOP720_FQ2;Write;SOP720_FQ2;Digital;;
CODESYSSPV3/3S/IecVarAccess;String;|var|CODESYS Control Win V3 x64.Application.IOs.SOP720_B2;Write;SOP720_B2;Digital;;
CODESYSSPV3/3S/IecVarAccess;String;|var|CODESYS Control Win V3 x64.Application.IOs.SOP720_B3;Write;SOP720_B3;Digital;;
CODESYSSPV3/3S/IecVarAccess;String;|var|CODESYS Control Win V3 x64.Application.IOs.SOP720_B8;Write;SOP720_B8;Digital;;
CODESYSSPV3/3S/IecVarAccess;String;|var|CODESYS Control Win V3 x64.Application.IOs.SOP720_HMI_B1;Write;SOP720_HMI_B1;Digital;;
CODESYSSPV3/3S/IecVarAccess;String;|var|CODESYS Control Win V3 x64.Application.IOs.SOP721_FQ1;Write;SOP721_FQ1;Digital;;
CODESYSSPV3/3S/IecVarAccess;String;|var|CODESYS Control Win V3 x64.Application.IOs.SOP721_B1;Write;SOP721_B1;Digital;;
CODESYSSPV3/3S/IecVarAccess;String;|var|CODESYS Control Win V3 x64.Application.IOs.SOP730_FQ1;Write;SOP730_FQ1;Digital;;
CODESYSSPV3/3S/IecVarAccess;String;|var|CODESYS Control Win V3 x64.Application.IOs.SOP730_B1;Write;SOP730_B1;Digital;;
CODESYSSPV3/3S/IecVarAccess;String;|var|CODESYS Control Win V3 x64.Application.IOs.SOP730_B2;Write;SOP730_B2;Digital;;
CODESYSSPV3/3S/IecVarAccess;String;|var|CODESYS Control Win V3 x64.Application.IOs.SOP730_B3;Write;SOP730_B3;Digital;;
CODESYSSPV3/3S/IecVarAccess;String;|var|CODESYS Control Win V3 x64.Application.IOs.SOP722_FQ1;Write;SOP722_FQ1;Digital;;
CODESYSSPV3/3S/IecVarAccess;String;|var|CODESYS Control Win V3 x64.Application.IOs.SOP722_B1;Write;SOP722_B1;Digital;;
CODESYSSPV3/3S/IecVarAccess;String;|var|CODESYS Control Win V3 x64.Application.IOs.SOP723_FQ1;Write;SOP723_FQ1;Digital;;
CODESYSSPV3/3S/IecVarAccess;String;|var|CODESYS Control Win V3 x64.Application.IOs.SOP723_B1;Write;SOP723_B1;Digital;;
CODESYSSPV3/3S/IecVarAccess;String;|var|CODESYS Control Win V3 x64.Application.IOs.SOP723_HMI_B1;Write;SOP723_HMI_B1;Digital;;
CODESYSSPV3/3S/IecVarAccess;String;|var|CODESYS Control Win V3 x64.Application.IOs.SOP720_HMI_B2;Write;SOP720_HMI_B2;Digital;;
CODESYSSPV3/3S/IecVarAccess;String;|var|CODESYS Control Win V3 x64.Application.IOs.SOP723_HMI_B2;Write;SOP723_HMI_B2;Digital;;
CODESYSSPV3/3S/IecVarAccess;String;|var|CODESYS Control Win V3 x64.Application.IOs.SOP720_B9;Write;SOP720_B9;Digital;;
CODESYSSPV3/3S/IecVarAccess;String;|var|CODESYS Control Win V3 x64.Application.IOs.SOP713_B4;Write;SOP713_B4;Digital;;
CODESYSSPV3/3S/IecVarAccess;String;|var|CODESYS Control Win V3 x64.Application.IOs.SOP713_B5;Write;SOP713_B5;Digital;;
CODESYSSPV3/3S/IecVarAccess;String;|var|CODESYS Control Win V3 x64.Application.IOs.SOP730_B4;Write;SOP730_B4;Digital;;
CODESYSSPV3/3S/IecVarAccess;String;|var|CODESYS Control Win V3 x64.Application.IOs.SOP730_B5;Write;SOP730_B5;Digital;;
CODESYSSPV3/3S/IecVarAccess;String;|var|CODESYS Control Win V3 x64.Application.IOs.SOP720_LC1_ON;Write;SOP720_LC1_ON;Digital;;
CODESYSSPV3/3S/IecVarAccess;String;|var|CODESYS Control Win V3 x64.Application.IOs.SOP720_LC2_ON;Write;SOP720_LC2_ON;Digital;;
CODESYSSPV3/3S/IecVarAccess;String;|var|CODESYS Control Win V3 x64.Application.IOs.SOP723_LC1_ON;Write;SOP723_LC1_ON;Digital;;
CODESYSSPV3/3S/IecVarAccess;String;|var|CODESYS Control Win V3 x64.Application.IOs.SOP723_LC2_ON;Write;SOP723_LC2_ON;Digital;;
CODESYSSPV3/3S/IecVarAccess;String;|var|CODESYS Control Win V3 x64.Application.IOs.SOP720_Dispensed;Write;SOP720_Dispensed;Digital;;
CODESYSSPV3/3S/IecVarAccess;String;|var|CODESYS Control Win V3 x64.Application.IOs.Box_MB16_Acc;Read;Box_MB16_Acc;Digital;;
CODESYSSPV3/3S/IecVarAccess;String;|var|CODESYS Control Win V3 x64.Application.IOs.Box_MB16T_Acc;Read;Box_MB16T_Acc;Digital;;
CODESYSSPV3/3S/IecVarAccess;String;|var|CODESYS Control Win V3 x64.Application.IOs.Box_MB20_Acc;Read;Box_MB20_Acc;Digital;;
CODESYSSPV3/3S/IecVarAccess;String;|var|CODESYS Control Win V3 x64.Application.IOs.Box_MB24_Acc;Read;Box_MB24_Acc;Digital;;
CODESYSSPV3/3S/IecVarAccess;String;|var|CODESYS Control Win V3 x64.Application.IOs.Box_MB16_Rej;Read;Box_MB16_Rej;Digital;;
CODESYSSPV3/3S/IecVarAccess;String;|var|CODESYS Control Win V3 x64.Application.IOs.Box_MB16T_Rej;Read;Box_MB16T_Rej;Digital;;
CODESYSSPV3/3S/IecVarAccess;String;|var|CODESYS Control Win V3 x64.Application.IOs.Box_MB20_Rej;Read;Box_MB20_Rej;Digital;;
CODESYSSPV3/3S/IecVarAccess;String;|var|CODESYS Control Win V3 x64.Application.IOs.Box_MB24_Rej;Read;Box_MB24_Rej;Digital;;
CODESYSSPV3/3S/IecVarAccess;String;|var|CODESYS Control Win V3 x64.Application.IOs.Pallet_Creation;Read;Pallet_Creation;Digital;;
CODESYSSPV3/3S/IecVarAccess;String;|var|CODESYS Control Win V3 x64.Application.IOs.SOP710_KM1;Read;SOP710_KM1;Digital;;
CODESYSSPV3/3S/IecVarAccess;String;|var|CODESYS Control Win V3 x64.Application.IOs.SOP710_KM2;Read;SOP710_KM2;Digital;;
CODESYSSPV3/3S/IecVarAccess;String;|var|CODESYS Control Win V3 x64.Application.IOs.SOP711_KM1;Read;SOP711_KM1;Digital;;
CODESYSSPV3/3S/IecVarAccess;String;|var|CODESYS Control Win V3 x64.Application.IOs.SOP711_KM2;Read;SOP711_KM2;Digital;;
CODESYSSPV3/3S/IecVarAccess;String;|var|CODESYS Control Win V3 x64.Application.IOs.SOP712_KM1;Read;SOP712_KM1;Digital;;
CODESYSSPV3/3S/IecVarAccess;String;|var|CODESYS Control Win V3 x64.Application.IOs.SOP712_KM2;Read;SOP712_KM2;Digital;;
CODESYSSPV3/3S/IecVarAccess;String;|var|CODESYS Control Win V3 x64.Application.IOs.SOP713_KM1;Read;SOP713_KM1;Digital;;
CODESYSSPV3/3S/IecVarAccess;String;|var|CODESYS Control Win V3 x64.Application.IOs.SOP713_KM2;Read;SOP713_KM2;Digital;;
CODESYSSPV3/3S/IecVarAccess;String;|var|CODESYS Control Win V3 x64.Application.IOs.SOP713_K3;Read;SOP713_K3;Digital;;
CODESYSSPV3/3S/IecVarAccess;String;|var|CODESYS Control Win V3 x64.Application.IOs.SOP713_K4;Read;SOP713_K4;Digital;;
CODESYSSPV3/3S/IecVarAccess;String;|var|CODESYS Control Win V3 x64.Application.IOs.SOP713_K5;Read;SOP713_K5;Digital;;
CODESYSSPV3/3S/IecVarAccess;String;|var|CODESYS Control Win V3 x64.Application.IOs.SOP713_K6;Read;SOP713_K6;Digital;;
CODESYSSPV3/3S/IecVarAccess;String;|var|CODESYS Control Win V3 x64.Application.IOs.SOP714_KM1;Read;SOP714_KM1;Digital;;
CODESYSSPV3/3S/IecVarAccess;String;|var|CODESYS Control Win V3 x64.Application.IOs.SOP714_KM2;Read;SOP714_KM2;Digital;;
CODESYSSPV3/3S/IecVarAccess;String;|var|CODESYS Control Win V3 x64.Application.IOs.SOP715_KM1;Read;SOP715_KM1;Digital;;
CODESYSSPV3/3S/IecVarAccess;String;|var|CODESYS Control Win V3 x64.Application.IOs.SOP715_KM2;Read;SOP715_KM2;Digital;;
CODESYSSPV3/3S/IecVarAccess;String;|var|CODESYS Control Win V3 x64.Application.IOs.SOP716_KM1;Read;SOP716_KM1;Digital;;
CODESYSSPV3/3S/IecVarAccess;String;|var|CODESYS Control Win V3 x64.Application.IOs.SOP716_KM2;Read;SOP716_KM2;Digital;;
CODESYSSPV3/3S/IecVarAccess;String;|var|CODESYS Control Win V3 x64.Application.IOs.SOP717_KM1;Read;SOP717_KM1;Digital;;
CODESYSSPV3/3S/IecVarAccess;String;|var|CODESYS Control Win V3 x64.Application.IOs.SOP717_KM2;Read;SOP717_KM2;Digital;;
CODESYSSPV3/3S/IecVarAccess;String;|var|CODESYS Control Win V3 x64.Application.IOs.SOP720_KM1;Read;SOP720_KM1;Digital;;
CODESYSSPV3/3S/IecVarAccess;String;|var|CODESYS Control Win V3 x64.Application.IOs.SOP720_KM2;Read;SOP720_KM2;Digital;;
CODESYSSPV3/3S/IecVarAccess;String;|var|CODESYS Control Win V3 x64.Application.IOs.SOP720_KM3;Read;SOP720_KM3;Digital;;
CODESYSSPV3/3S/IecVarAccess;String;|var|CODESYS Control Win V3 x64.Application.IOs.SOP720_KM4;Read;SOP720_KM4;Digital;;
